	(* Flags to trigger the alarms/events *) //--------------------------------------------------------------------
	
	aSolventLowLevel	 : ARRAY[1..4] OF BOOL; //Flags to check the solvent levels before going to auto cycle
	aSolventNearLowLevel : ARRAY[1..4] OF BOOL; //Flags to warning if the solvent levels are near low level
	bWasteHighLevel		 : BOOL; //Flag to check waste reservoir level before going to auto cycle
	bWasteNearHighLevel	 : BOOL; //Flag to warning if waste reservoir is new high level
	
	bPumpsEStopTriggered : BOOL; //Flag when pumps were running and a emergency stop is triggered
	
	rDiskUsage_C : LREAL;   // % Percentage usage of C: on IPC hard drive
	
	bTCPCLientConnectError	: BOOL; // TCP Client FB_SocketConnect error Flag
	bTCPCLientSendError		: BOOL; // TCP Client FB_SocketSend error Flag
	bTCPCLientReceiveError	: BOOL; // TCP Client FB_SocketReceive error Flag
	bTCPCLientCloseError	: BOOL; // TCP Client FB_SocketCloseAll or FB_SocketClose error Flag
 
	bInvalidSolventSelection : BOOL; // Calibration Invalid Solvent Selection Error
	sStartCalibrationBlockedReason : STRING(255); // Calibration Invalid Solvent Selection Reason
	
	(* Motion Timeouts *) //---------------------------------------------------------------------------------------
	//System Init
	bMotionResetTimeout		: BOOL;	// Motion Timeout during Reset step on PRG_SystemInit
	bMotionEnableTimeout	: BOOL; // Motion Timeout during Enable step on PRG_SystemInit
	bMotionHomeTimeout		: BOOL; // Motion Timeout during Homing step on PRG_SystemInit
	bMotionMoveAbsTimeout	: BOOL; // Motion Timeout during Move Absolute step on PRG_SystemInit
	
	sMotionResetTimeoutAxis		: STRING(64); // String including the axis names to be part of alarm text - Motion Timeout during Reset step on PRG_SystemInit
	sMotionEnableTimeoutAxis	: STRING(64); // String including the axis names to be part of alarm text - Motion Timeout during Enable step on PRG_SystemInit
	sMotionHomeTimeoutAxis		: STRING(64); // String including the axis names to be part of alarm text - Motion Timeout during Homing step on PRG_SystemInit
	sMotionMoveAbsTimeoutAxis	: STRING(64); // String including the axis names to be part of alarm text - Motion Timeout during Move Absolute step on PRG_SystemInit
	
	(* Secondary Functions *) //---------------------------------------------------------------------------------------
	bCalJsonCreationError		: BOOL;		// Error during calibration json file creation
	nCalJsonCreationErrorId		: UDINT;	// Error number ID during calibration json file creation
	
END_VAR

// ---- GVLs/GVL_Calibration.TcGVL
{attribute 'qualified_only'}
VAR_GLOBAL
	
	aCalibPumps         : ARRAY[1..10] OF ST_CalibrationPump;
    bStartCalibration   : BOOL;
    bAbortCalibration   : BOOL;
    bCalibrationRunning : BOOL;
    bCalibrationDone    : BOOL;
    eCalibSolvent       : E_SolventType;
    tDelayStart         : TIME;
    bPrintWhenComplete  : BOOL;
    sGlobalStatus       : STRING[100];
	iPercentLoadBar     : UINT;
	iReplicatesSetpoint : UINT := 1; 
	rAcceptanceCriteria	: LREAL;
	iAllowableFailures	: UINT := 2;
	fbScaleDevice		: FB_ScaleDevice; //Scale Instance Object
	iResultIndex	 	: INT;		 	// Array index on calibration results
	
	aCalibLinearPumps	: ARRAY[1..10] OF ST_LinearPumpCalibration;
	eLeakTestState 		: E_LeakTestState	:= E_LeakTestState.IDLE;
	
	// temp 
	aDosingResults		: ARRAY[1..50] OF ST_DosingResults;
	
	//aCalibCheckResult	: ARRAY[1..100] OF ST_CalibrationPumpResult;
	
	(* Calibration Report*)// -----------------------------------------------------------------------------------------------
	//																													 	|
	stPumpCalReportInfo 	: ST_ReportInfo;	  	//																	  	|
	stPumpCalibrationInfo 	: ST_CalibrationInfo;	//																		|
	stPumpCalibrationData 	: ARRAY[1..250] OF ST_CalibrationData;	//
	//																	
	stLinearCalibrationData : ARRAY[1..10] OF ST_LinearPumpControllDB; // Linear Calibration changing position data from HMI
	//																														|		
	bStartCreationCalJson	: BOOL; // Flag to start the Json creation														|
	bCreationCalJsonDone	: BOOL; // Flag to indicate Json was created Correctly											|
	bCreationCalJsonError	: BOOL; // Flag to indicate Error on Json creation												|
	//																														|
	(**)//-------------------------------------------------------------------------------------------------------------------
	
	//Dosing Procedure
	bDosingTestEnable : BOOL := FALSE;
	
END_VAR

// ---- GVLs/GVL_Constant.TcGVL
{attribute 'qualified_only'}
VAR_GLOBAL CONSTANT

(*Calibration Reports Info*) //----------------------------------------------------------------------------------------------------------------------------
sPumpCalibrationReportName		: STRING(64) := 'Tegan Automated Sample Recovery System (ASRS)';
sPumpCalibrationReportSubName	: STRING(64) := 'Pump Calibration Report';
sSystemID						: STRING(16) := '0001';
sDatabaseName					: STRING(16) := 'ASRS_25';

(*Solvents Types into screen combo boxes*) //--------------------------------------------------------------------------------------------------------------
aSolventsAvailable : ARRAY[1..5] OF STRING := [ 'Solvent 1' , 'Solvent 2', 'Solvent 3', 'Solvent 4', 'Solvent 5' ];

(*IO Screen Texts and pages*) //---------------------------------------------------------------------------------------------------------------------------
aIOPageStarts : ARRAY[0..20] OF UDINT  := [ 0, 1, 3, 5, 7, 9, 11, 13, 15, 17, 19, 21, 23, 25, 27, 29, 31, 33, 35, 37, 40];

aIOList		  :	ARRAY[0..42] OF STRING := [	'  System Overview',
											'  Beckhoff C6030-0060 | Ultra-Compact Industrial PC',
											'  Beckhoff CP2921-0000 | Multi-touch Built-in Control Panel',
											'  Term 1 : EK1100 | EtherCAT Coupler',
											'  Term 2 : EL6070-0033 | License Key Terminal for TwinCAT 3.1',
											
											'  Term 3 : EL6910 | TwinSAFE PLC Module',
											
											'  Term 4 : EL1918 | 8-Channel Digital Input Terminal, TwinSAFE',
											'  Term 5 : EL1918 | 8-Channel Digital Input Terminal, TwinSAFE',
											'  Term 6 : EL1918 | 8-Channel Digital Input Terminal, TwinSAFE',
											
											'  Term 7 : EL2904 | 4-Channel Digital Output Terminal, TwinSAFEE',
											'  Term 8 : EL2904 | 4-Channel Digital Output Terminal, TwinSAFE',
											
											'  Term 9 : EL1809 | 16-Channel Digital Input Terminal',
											'  Term 10: EL2809 | 16-Channel Digital Output Terminal',
											
											'  Term 11: EL2624 | 4-channel Relay Output Terminal',
											
											'  Term 12: EL9410 | Power supply terminal for E-bus, with diagnostics',
											'  Term 13: EL3058 | 8-channel analog input, current, single-ended',
											'  Term 14: EL9576 | Brake chopper terminal',
											'  Term 15: EL7211-9014 | 1-channel Motion interface, servomotor',
											'  Term 16: EL7211-9014 | 1-channel Motion interface, servomotor',
											'  Term 17: EL3022 | 2-channel analog input, current, differential',
											'  Term 18: EL1809 | 16-channel digital input, 24 V DC, 3 ms',
											'  Term 19: EL2904 | 4-Channel Digital Output Terminal, TwinSAFE',
											'  Term 20: EL6631 |  2-port Communication PROFINET RT Interface',					
											
											'  Term 22: EL7062 | 2-channel Motion Stepper Motor Interface',
											'  Term 23: EL7062 | 2-channel Motion Stepper Motor Interface',
											'  Term 24: EL7062 | 2-channel Motion Stepper Motor Interface',
											'  Term 25: EL7062 | 2-channel Motion Stepper Motor Interface',
											'  Term 26: EL7062 | 2-channel Motion Stepper Motor Interface',
											'  Term 27: EL7062 | 2-channel Motion Stepper Motor Interface',
											'  Term 28: EL7062 | 2-channel Motion Stepper Motor Interface',
											'  Term 29: EL7062 | 2-channel Motion Stepper Motor Interface',
											'  Term 30: EL7062 | 2-channel Motion Stepper Motor Interface',
											'  Term 31: EL7062 | 2-channel Motion Stepper Motor Interface',
											'  Term 32: EL7062 | 2-channel Motion Stepper Motor Interface',
											'  Term 33: AX8101 | Single-axis Module',
											
											'  BOX 01  - AL1333 | IO-Link master with EtherCAT interface',
											'  BOX 02 - AMI8100 | Compact Integrated Servo Drives',	
											'  BOX 03 - AMI8100 | Compact Integrated Servo Drives',		
											'  BOX 04 - AMI8100 | Compact Integrated Servo Drives',
											'  BOX 05 - AMI8100 | Compact Integrated Servo Drives',	
											'  BOX 06 - AMI8100 | Compact Integrated Servo Drives'			
											];

//Naming the axis by index for alarms text assemble
sMotionText	: ARRAY[1..28] OF STRING(5) := [ 'M1,',
											 'M2,',
											 'M3,',
											 'V1,',
											 'V2,',
											 'V3,',
											 'V4,',
											 'V5,',
											 'LP1,',
											 'LP2,',
											 'LP3,',
											 'LP4,',
											 'LP5,',
											 'LP6,',
											 'LP7,',
											 'LP8,',
											 'LP9,',
											 'LP10,',
											 'RP1,',
											 'RP2,',
											 'RP3,',
											 'RP4,',
											 'RP5,',
											 'RP6,',
											 'RP7,',
											 'RP8,',
											 'RP9,',
											 'RP10,'
 											];


(* ----------------------------------------------------------------------------------- HMI COLORS ----------------------------------------------------------------------------------- *)
	
    sWHITE                              :   STRING(40)  := '{"color":"rgba(255,255,255,255)"}';
    sBLACK                              :   STRING(40)  := '{"color":"rgba(0,0,0,1)"}';
    sYELLOW                             :   STRING(40)  := '{"color":"rgba(255,255,0,1)"}';
    sGREEN                             	:   STRING(40)  := '{"color":"rgba(70,166,63,1)"}';
	sLGREEN                             :   STRING(40)  := '{"color":"rgba(58,211,20,1)"}';
    sORANGE                             :   STRING(40)  := '{"color":"rgba(255,153,51,1)"}';
    sNYPROORANGE                        :   STRING(40)  := '{"color":"rgba(255,140,0,1)"}';
    sRED                                :   STRING(40)  := '{"color":"rgba(255,0,0,1)"}';
	sLRED                               :   STRING(40)  := '{"color":"rgba(233,53,44,1)"}';
    sBLUE                               :   STRING(40)  := '{"color":"rgba(0,0,255,1)"}';
	sLBLUE                              :   STRING(40)  := '{"color":"rgba(0,162,232,1)"}';
    sGREY                               :   STRING(40)  := '{"color":"rgba(164,158,158,1)"}';
    sScreenGREY                         :   STRING(40)  := '{"color":"rgba(225,225,225,1)"}';
    sDARKGREY                           :   STRING(40)  := '{"color":"rgba(50,50,50,1)"}';
    sPURPLE                             :   STRING(40)  := '{"color":"rgba(128,0,128,1)"}';
    sVIOLET                             :   STRING(40)  := '{"color":"rgba(204,153,255,1)"}';
    sTRANSP                             :   STRING(40)  := '{"color":"rgba(255,255,255,0)"}';
    sGREENPass                          :   STRING(40)  := '{"color":"rgba(0,153,51,1)"}';
    sREDFail                            :   STRING(40)  := '{"color":"rgba(244,68,68,255)"}';
    sBLUEInProgress                     :   STRING(40)  := '{"color":"rgba(54,100,221,1)"}';
	sGREENISHTEAColor					:	STRING(40)  := '{"color":"rgba(60,192,134,255)"}'	;		

	nBLACK								: 	DWORD 	:= 	16#FF000000;	 // format: TTRRGGBB where T -> 00 = full transparency and FF = full opaque
	nWHITE								: 	DWORD 	:= 	16#FFFFFFFF;
	nYELLOW								: 	DWORD 	:= 	16#FFFFFF00; 
	nGREEN								: 	DWORD 	:= 	16#FF008A00;
	nLIGHTGREEN                         :   DWORD   :=  16#FF98FB89;
	nORANGE								: 	DWORD 	:= 	16#FFFFA500;
	nNYPROORANGE						:	DWORD	:=	16#FFF05322;
	nRED								: 	DWORD 	:= 	16#FFFF0000;
	nBLUE								: 	DWORD 	:= 	16#FF0000FF;
	nLIGHTBLUE                          :   DWORD   :=  16#FF08ADF4;
	nGREY								: 	DWORD 	:= 	16#FFA9A9A9;	
	nDARKGREY							:	DWORD	:=	16#FF808080;
	nPURPLE								:	DWORD	:=	16#FF800080;
	nVIOLET								:	DWORD	:=	16#FFEE82EE;
	nTRANSP								:	DWORD	:=	16#00FFFFFF;	// full transparent WHITE
	
(* ----------------------------------------------------------------------------------- HMI COLORS ----------------------------------------------------------------------------------- *)
											
END_VAR

// ---- GVLs/GVL_HMI.TcGVL
{attribute 'qualified_only'}
{attribute 'TcHmiSymbol' := 'true'}
VAR_GLOBAL
	
	//Info Screen
	stInfo				: ST_InfoPage; 	// Project Info screen details to be shown on HMI
	stReminders 		: ST_Reminders; // Reminders screen signals to be shown on HMI
	
	HMIDigInputs		 : ST_HMIDigInputs;  //Digital Inputs data from HMI
	HMIDigOutputs		 : ST_HMIDigOutputs; //Digital Outputs data for HMI

	HMIAnimation		 : ST_HMIAnimation; //Variables needed to animate the HMI
	bHMICalibrationBox	 : BOOL; 			//Calibration Box presence
	
	eMachineMode		 : E_MachineMode; //Machine mode selection from HMI
	
	bIncoherenceDetected : BOOL := FALSE; //Incoherence Monitoring that could block master controll to enter in autoCycle
	bIncoherenceAlert	 : BOOL := FALSE; //Incoherence alert to show an alert on HMI. Event trigger DesktopView 
	
	sDateAndTimeEventTriggered	: STRING(256); //Linear Pumps save procedure gets the date and time from hmi
	sUserNameEventTriggered		: STRING(256); //Linear Pumps save procedure gets the hmi username
	
	sActivatedRecipeHomeNaming  : STRING(256); // Recipe name shown on home screen when a recipe is active
	
	(* Auto Cycle Popup *) // ---------------------------------------------------------------------------------------------------------------------------------
	sAutoCycleComment			: STRING(256); // Comment inserted by user before going to autocycle
	bStartAutoCycleButton		: BOOL := FALSE; // Start AUto Cycle Button from Auto Cycle popup
	bShowAutoCyclePopup     	: BOOL := FALSE; // Controls Auto Cycle popup visibility on HMI
	bSystemReady_ReqAutoCycle 	: BOOL := FALSE; // One-shot request to go to AUTO_CYCLE from SystemReady
	
	// --- Auto cycle soft-stop / hold control ---
    bAutoCycleHoldReq        : BOOL	:= FALSE;  // 1st STOP inside AUTO_CYCLE
    bAutoCycleHoldActive     : BOOL	:= FALSE;  // TRUE while StateMachine is in PAUSE_STATE
    bAutoCycleHoldPopup      : BOOL := FALSE;  // HMI shows the "Cancel / Continue" popup
	bAutoCyclePrimeSolvents	 : BOOL	:= FALSE;  // HMI flag for prime the solvents used on auto cycle before metering the rinse

    bAutoCycleContinueCmd    : BOOL	:= FALSE;  // HMI "Continue" button
    bAutoCycleCancelCmd      : BOOL	:= FALSE;  // HMI "Cancel Run" button
	
	bLightsToggleButton	 : BOOL := FALSE; // Home screen toggle button for turn lights on or off on HMI 
	rTimeCountingDown 	 : LREAL; 		  //Countdown time for shutdown or rebooting PLC
	sCountdownPopupText	 : STRING(16);	  //Countdown Popup text for shutdown or rebooting PLC
	
	//Machine Mode Blinking
	bMachineModeBlinking : BOOL := FALSE;	// Flashing variable to blink the state on HMI headbar
	bMachineModeScan	 : BOOL := FALSE;	// Flashing variable to scan some controls on HMI home screen
	bHomeScreenLoaded	 : BOOL := FALSE;	// Flag to tell when the home screen is loaded or not
	
	//User Management
	stUserMgmtHistoryEvent  : ST_UserMgmtHistoryEvent;
	stUsers          		: ARRAY[1..50] OF ST_User;  // users list | max 50 users
    iLoggedUserID    		: INT := -1;                // -1 = no one logged in
    dtCurrentLogin   		: DT;
    tSessionStart    		: TIME;

	// <Recipe> Variables needed to handle recipe --------------------------------------------------------------------------------------------------------------
	aAvailableFiles         : ARRAY[0..99] OF ST_RecipeFileInfo;
    iFileCount              : INT;
	
    bRefreshRecipeList      : BOOL; 			//List the recipe files from HMI
    bRecipeLoadFromFile	 	: BOOL := FALSE; 	//load recipe button from HMI
	bReloadRecipeDatagrids	: BOOL := FALSE;	//Reload the recipe in stCurrentRecipe to the datagrids if the cancel button is pressed when creating new recipe
    sSelectedRecipeName     : STRING(255); 		// Selected name from hmi list popup
	bRecipeCorrectLoaded	: BOOL; 			// Flag to identify if there is a recipe loaded to proceed with the recovery
	bRecipeLoadFailed		: BOOL; 			// Flag to identify if there was any error loading the recipe file
	
	bRecipeActivateButton	: BOOL := FALSE; // Activate Recipe command from recipe activate button 
	bRecipeActivateDone		: BOOL := FALSE; // Activate done flag after command from recipe activate button
	bRecipeActivateError	: BOOL := FALSE; // Activate Error flag after command from recipe activate button
	
	bRecipeSaveButton		: BOOL := FALSE; // save command from recipe save button
	bRecipeSaveDone			: BOOL := FALSE; // Save done flag after save command from recipe save button
	bRecipeSaveError		: BOOL := FALSE; // Save Error flag after save command from recipe save button
	
	stDeleteRecipeInfo		: ST_RecipeFileInfo;
	bDeleteRecipeButton		: BOOL := FALSE; // Delete recipe button Action - Open delete popup
	bDeleteRecipeConfirm	: BOOL := FALSE; // Delete recipe confirmation action
	bDeleteRecipeError		: BOOL := FALSE; // Delete recipe Error flag
	bDeleteRecipeDone		: BOOL := FALSE; // Delete recipe done flag
	
	bNewRecipeButton		: BOOL := FALSE; // New Recipe button on recipe screen.
	
	//Recipe HMI View - data needs to be transposed for better view and handled by HMI
	stRecipeInfo		 : ST_RecipeInfo;	// Recipe info datagrid showed on HMI
	aSolventAndTimesRows : ARRAY[1..3] OF ST_HMI_SolventAndTimeRow;	// Recipe Solvent And Times transposed datagrid showed on HMI
	aVolumeRows 		 : ARRAY[1..10] OF ST_HMI_VolumesRow; 		// Recipe Volumes transposed datagrid showed on HMI
	aOtherParamsRows 	 : ARRAY[1..8] OF ST_HMI_OtherParamsRow;	// Recipe Other Parameters transposed datagrid showed on HMI
	// <\Recipe> -----------------------------------------------------------------------------------------------------------------------------------------------
	
	// <Calibration> Variables needed to handle calibration tasks from HMI -------------------------------------------------------------------------------------
	
	bCalLeakTestButton		: BOOL := FALSE; // Leak test action button from HMI
	bCalLeakTestPass		: BOOL := FALSE; // Leak test passed flag
	bCalLeakTestFail		: BOOL := FALSE; // Leak test failed flag
	bCalLeakTestError		: BOOL := FALSE; // Leak test error flag
	rCalLeakTestPressure	: LREAL;		 // Leak test pressure reading from sensor
	
	bCalPressureUpSystemBt	: BOOL := FALSE; // HMI Button responsible for pressurize the system
	bCalHoldSysPressureBt	: BOOL := FALSE; // HMI Button responsible for shut the air off the system
	bCalStopLeakTestBt		: BOOL := FALSE; // HMI Button responsible for stopping the leak test
	
	bCalLinearPumpsEnableBt	: BOOL := FALSE; // Linear pumps Enable motors button
	bCalLinearPumpsHomeBt	: BOOL := FALSE; // Linear pumps Homing motors button
	bCalLinearPumpsMoveBt	: BOOL := FALSE; // Linear pumps Move motors button
	bCalLinearPumpsStopBt	: BOOL := FALSE; // Linear pumps Stop motors button
	bCalLinearPumpsSaveBt	: BOOL := FALSE; // Linear pumps Save Parameters button
	bCalLinearPumpsDirty	: BOOL := FALSE; // flag to indicate when there was any change on the linear pumps.
	
	bStartCalibrationBt		: BOOL := FALSE; //Start Calibration Bt from HMI
	bAbortCalibrationBT		: BOOL := FALSE; //Abort Calibration Bt from HMI
	
	aCalibPumps         	: ARRAY[1..10] OF ST_CalibrationPump;		// Calibration rotary Pumps settings
	aCalibLinearPumps		: ARRAY[1..10] OF ST_LinearPumpCalibration; // Calibration linear Pumps settings
	aCalPumpResults    		: ARRAY[1..10] OF ST_CalibrationPumpResult; // Rotary Pumps result structure
	
	iSelectedCalibrationSolvent : USINT := 0; // Solvent Selection - 0 = None, 1 = Solvent 1, 2 = Solvent 2, etc.
	
	rLinearPumpsLastAdjustUser	: STRING(128);		 // Linear pumps last adjusted username
	rLinearPumpsLastAdjustDate	: DATE;				 // Linear pumps last adjusted Date
	
	bScaleNeedsAtention		: BOOL := FALSE; // Flag to trigger a popup on hmi telling operator to handle the scale error | Listener on Desktop.view Index Region
	bScaleFixed				: BOOL := FALSE; // Feedback from hmi to tell the system that scale is ready to continue
	
	bCalBoxNeedsAttention	: BOOL := FALSE; // Flag to trigger a popup on hmi telling operator to fill up the calibration box
	bCalBoxFixed			: BOOL := FALSE; // Feedback from hmi to tell the system that the calibration box is ready to continue
	
	bCalMoveValves			: BOOL  := FALSE; // Manual Valves Movement from calibration screen 
	iCalMoveValvesPosition	: USINT := 1; 	  // Manual Valves Position from calibration screen 
	bCalMoveM1Motor			: BOOL  := FALSE; // Manual M1 Motor Movement from calibration screen 
	iCalMoveM1MotorPosition	: USINT := 1; 	  // Manual M1 Motor Position from calibration screen 
	
	sCalLeakTestStatus		: STRING(32);	  // Automatic sealing test status text on calibration screen 
	iCalLeakTestState		: USINT := 1;	  // Automatic sealing test image state LED on calibration screen 
	
	//UILoadBar
	bCalibStepLoading   : BOOL;		  	// Loadbar progress enable variable on calibration screen
    rCalibStepPercent   : REAL;       	// Loadbar progress for step time on calibration screen [0..100]
    sCalibProgressLabel : STRING(80);	// Loadbar progress label on calibration screen
	
	// <\Calibration> ------------------------------------------------------------------------------------------------------------------------------------------
	
	// <Reports Listing> ---------------------------------------------------------------------------------------------------------------------------------------
	
	aCalibrationReportList      : ARRAY[1..100] OF ST_CalibrationReportListItem;
    stSelectedCalibReportHeader : ST_CalibrationReportHeader;
    aSelectedCalibReportLines   : ARRAY[1..300] OF ST_CalibrationReportLine;

    sSelectedReportId           : STRING(50);

    bLoadCalibrationReportList  : BOOL;
    bLoadSelectedCalibReport    : BOOL;
    bSelectedReportReady        : BOOL;
    bReportListReady            : BOOL;
    bReportQueryBusy            : BOOL;
    bReportQueryError           : BOOL;
	
	aReportSearchResult : ARRAY[1..100] OF ST_ReportListItem;
	uiReportSearchCount : UDINT;
	eSelectedReportType : E_ReportType;
	sSelectedPrimaryID  : STRING(50);
	dtDateFrom          : STRING(30);
	dtDateTo            : STRING(30);
	
	// <Machine Settings> Variables to handle solvents insert in the settings screen ----------------------------------------------------------------------------
	HMIParameters		 : ST_HMIParameters; 					// Motion Parameters from HMI inputs
	stHMICalibParameters : ST_CalibrationSettings;				// Calibration Parameters from HMI inputs
	stHMIPumpParameters	 : ST_PumpSettings;						// Pump Parameters from HMI inputs
	stLeakTestParameters : ST_LeakTestSettings;					// Leak Test Parameters from HMI Inputs
	stHMISolventsInfo	 : ARRAY[1..4] OF ST_SolventsSettings;	// Solvents name and density to be inserted on the settings screen 		
	bReloadHMIParameters : BOOL := FALSE;						// Reload parameters from GVL_Settings when first loading the screen
	bSaveParametersBt	 : BOOL := FALSE; 						// Save Parameters from HMI
	bSaveParametersDone	 : BOOL := FALSE;						// Save Parameters Done flag from PLC
 	bSaveParametersError : BOOL := FALSE;						// Save Parameters Error flag from PLC
	bSaveSolventsBt		 : BOOL := FALSE;						// Save Solvents change from HMI settings screen
	bSaveSolventsDone	 : BOOL := FALSE;						// Save Solvents Done flag from HMI settings screen
	bSaveSolventsError	 : BOOL := FALSE;						// Save Solvents Error flag from HMI settings screen
	
	(* Manual Motors Moviment *) //--------------------------------------------------------------------------------------------------------------
	ManualMov			: ST_MotorsJog; // Manual Joging motors from old manual screen
	
	aManualMotorsCmd 	: ARRAY[1..3] OF ST_MotorCommand;	// Manual Motors commands from manual screen
    aManualValvesCmd 	: ARRAY[1..5] OF ST_ValveCommand;	// Manual Valves commands from manual screen
    aManualPumpsCmd  	: ARRAY[1..10] OF ST_PumpCommand;	// Manual Pumps commands from manual screen
	
	bRunPumpsBySpeedBt 		: BOOL;	// Button Run pumps by Speed from manual screen
	bRunPumpsByVolumeBt 	: BOOL;	// Button Run pumps by Volume from manual screen
	bRunPumpsByDistanceBt 	: BOOL;	// Button Run pumps by Distance from manual screen
	bStopPumpsBt 			: BOOL;	// Button Stop pumps movememnt from manual screen
	
	(* Alarms and Events triggers from HMI JS Trigger*) //-------------------------------------------------------------------------------------------------------------
	bM1MoveNotAllowedTrigger	: BOOL;	// 'IE-100: M1 Movement Not allowed'; (* JS from Run M1 Button - Manual screen *)
	bM2MoveNotAllowedTrigger	: BOOL;	// 'IE-100: M2 Movement Not allowed'; (* JS from Run M2 Button - Manual screen *)
	bM3MoveNotAllowedTrigger	: BOOL;	// 'IE-101: M3 Movement Not allowed'; (* JS from Run M3 Button - Manual screen *)
	bCalNotAllowedTrigger		: BOOL;	// 'IE-110: Attempt to perform a calibration procedure without a calibration box'; (* JS from Start Calibration Button - Calibration screen *)
		
	// <IO Screen> Variables for IO Screen use (*-----------------------------------------------------------------------------------------------)
	
	nSelectedIO		: UDINT; // Selection made by IO screen combobox
	
	aIOTerm04		: ARRAY[1..8] OF BOOL;
	aIOTerm05		: ARRAY[1..8] OF BOOL; 
	aIOTerm06		: ARRAY[1..8] OF BOOL; 
	aIOTerm07		: ARRAY[1..4] OF BOOL; 
	aIOTerm08		: ARRAY[1..4] OF BOOL;
	aIOTerm09		: ARRAY[1..16] OF BOOL;
	aIOTerm10		: ARRAY[1..16] OF BOOL;
	aIOTerm11		: ARRAY[1..4] OF BOOL;   
	aIOTerm12		: ARRAY[1..2] OF BOOL;
	aIOTerm13		: ARRAY[1..8] OF REAL;
	aIOTerm14		: ARRAY[1..8] OF BOOL;
   	iIOTerm14DCIn	: UDINT;
	aIOTerm15		: ARRAY[1..3] OF BOOL;
	aIOTerm15Values : ARRAY[1..3] OF LREAL;
	iIOTerm15ErrorCode	: UDINT;
	aIOTerm16		: ARRAY[1..3] OF BOOL;
	aIOTerm16Values : ARRAY[1..3] OF LREAL;
	iIOTerm16ErrorCode	: UDINT;
	aIOTerm17		: ARRAY[1..6] OF BOOL;
	aIOTerm17Values : ARRAY[1..2] OF LREAL;
	aIOTerm18		: ARRAY[1..16] OF BOOL;
	aIOTerm19		: ARRAY[1..4] OF BOOL; 
	stIOTerm23		: ST_EL7062IOInfo;
	stIOTerm24		: ST_EL7062IOInfo;
	stIOTerm25		: ST_EL7062IOInfo;
	stIOTerm26		: ST_EL7062IOInfo;
	stIOTerm27		: ST_EL7062IOInfo;
	stIOTerm28		: ST_EL7062IOInfo;
	stIOTerm29		: ST_EL7062IOInfo;
	stIOTerm30		: ST_EL7062IOInfo;
	stIOTerm31		: ST_EL7062IOInfo;
	stIOTerm32		: ST_EL7062IOInfo;
	stIOTerm34		: ST_AX8101IOInfo;
	aIOBox1			: ARRAY[1..8] OF REAL;
	aIOAMI8000		: ARRAY[1..5] OF ST_AMI8000IOInfo;
	
	// <\IO Screen>  (*-------------------------------------------------------------------------------------------------------------------------)
	
	//TEMP
	bResetM1MotorBt : BOOL := FALSE; // Temporary Motor M1 Reset button on old joging manual screen while new motor is not installed
	
	// UserManagement -------------------------------------------------------------------------------------------------------------------
	
	passwordOk: BOOL;
	
END_VAR

// ---- GVLs/GVL_IO.TcGVL
{attribute 'qualified_only'}
VAR_GLOBAL
	
	(* IO used in the software *) //----------------------------------------------------------------------------------------
	gDigInputs	 		AT%I*	:	ST_EL1809;	//Digital inputs at Terminals 21 and 30 [EL1809]
	gDigOutputs			AT%Q*	:	ST_EL2809;	//Digital Outputs at Terminal 22 		[EL2809]
	gRelayOutputs		AT%Q*	:	ST_EL2624;	//Digital Relay Outputs at Terminal 23 	[EL2624]
	gAnalogInputs		AT%I*	:	ST_EL3058; 	//Analog inputs at Terminals 25 		[EL3058]
	gAnalogInputs2Ch	AT%I*	:	ST_EL3022;	//Analog inputs at Terminals 17 		[EL3022]
	gProfinetInput		AT%I*	:	ST_EL6631;  //Profinet inputs by Device 5 			[EL6631]
	
	gParameters			: ST_HMIParameters; 	//Machine Parameters
	gSetSolenoidControl : FB_SetSolenoid;		//FB only instance to control solenoids valves set. 
	
	// Safety Alias
	bInAckSignal		AT %I* : BOOL; // Aknowledge input
	bInResetSignal		AT %Q* : BOOL; // Reset input
	
	stEL6910	: ST_EL6910; // Safety PLC - Terminal 3
	
	// Is Vials Rack Present?
	bVialRackPresent : BOOL;
	
	// power source signal for recovery valves position purposes
	bPowerSupplyDropSignal	: BOOL := FALSE;
	
	//----------------------------------------------------------------------------------------------------------------------
	// IO Terminals to feed HMI IO Screens
	//----------------------------------------------------------------------------------------------------------------------
	
	// TERMINAL - EK1100 EtherCAT Coupler (Term 1)
	nEK1100T01State		AT %I*	: UINT;	//Terminal State from IO Terminal Info Data	
	bEK1100T01State				: BOOL; //Control flag from terminal state	
	sEK1100T01Status			: STRING(200);
	
	// TERMINAL - EK1100 EtherCAT Coupler (Term 22)
	nEK1100T22State		AT %I*	: UINT;	//Terminal State from IO Terminal Info Data
	bEK1100T22State				: BOOL; //Control flag from terminal state	
	sEK1100T22Status			: STRING(200);	
	
	// TERMINAL - EL6070-0033	License Key Terminal for TwinCAT 3.1 (Term 2)
	nEL6070State		AT %I*	: UINT;	// EL6070-0033 State from IO Terminal Info Data	
	bEL6070State				: BOOL; //Control flag from terminal state	
	sEL6070Status				: STRING(200);	
	
	// TERMINAL - EL1918 Safety Inputs (Term 4)
	nEL1918T04State		AT %I*	: UINT;	// EL1918 State from IO Terminal Info Data
	bEL1918T04State				: BOOL; //Control flag from terminal state		
	sEL1918T04Status			: STRING(200);	
	
	// TERMINAL - EL1918 Safety Inputs (Term 5)
	nEL1918T05State		AT %I*	: UINT;	// EL1918 State from IO Terminal Info Data
	bEL1918T05State				: BOOL; //Control flag from terminal state		
	sEL1918T05Status			: STRING(200);

	// TERMINAL - EL1918 Safety Inputs (Term 6)
	nEL1918T06State		AT %I*	: UINT;	// EL1918 State from IO Terminal Info Data	
	bEL1918T06State				: BOOL; //Control flag from terminal state	
	sEL1918T06Status			: STRING(200);	
	
	// TERMINAL - EL2904 Safety Outputs (Term 7)
	nEL2904T07State		AT %I*	: UINT;	// EL2904 State from IO Terminal Info Data
	bEL2904T07State				: BOOL; //Control flag from terminal state		
	sEL2904T07Status			: STRING(200);
	
	// TERMINAL - EL2904 Safety Outputs (Term 8)
	nEL2904T08State		AT %I*	: UINT;	// EL2904 State from IO Terminal Info Data	
	bEL2904T08State				: BOOL; //Control flag from terminal state	
	sEL2904T08Status			: STRING(200);
	
	// TERMINAL - EL1809 Digital Inputs (Term 9)
	nEL1809T09State		AT %I*	: UINT;	// State from IO Terminal Info Data	
	bEL1809T09State				: BOOL; // Control flag from terminal state	
	sEL1809T09Status			: STRING(200);
	
	// TERMINAL - EL2809 Digital Outputs (Term 10)
	nEL2809T10State		AT %I*	: UINT;	// State from IO Terminal Info Data	
	bEL2809T10State				: BOOL; // Control flag from terminal state	
	sEL2809T10Status			: STRING(200);
	
	// TERMINAL - EL2624 Relay Outputs (Term 11)
	nEL2624T11State		AT %I*	: UINT;	// State from IO Terminal Info Data	
	bEL2624T11State				: BOOL; // Control flag from terminal state	
	sEL2624T11Status			: STRING(200);
	
	// TERMINAL - EL9410 Power Supply (Term 12)
	nEL9410T12State		AT %I*	: UINT;	// State from IO Terminal Info Data	
	bEL9410T12State				: BOOL; // Control flag from terminal state	
	sEL9410T12Status			: STRING(200);
	bEL9410UPStatus		AT %I*	: BOOL; // Terminal UP Status
	bEL9410USStatus		AT %I*	: BOOL; // Terminal US Status
	
	// TERMINAL - EL3058 Relay Outputs (Term 13)
	nEL3058T13State		AT %I*	: UINT;	// State from IO Terminal Info Data	
	bEL3058T13State				: BOOL; // Control flag from terminal state	
	sEL3058T13Status			: STRING(200);
	
	// TERMINAL - EL9576 Relay Outputs (Term 14)
	nEL9576T14State			AT %I*	: UINT;	// State from IO Terminal Info Data	
	bEL9576T14State					: BOOL; // Control flag from terminal state	
	sEL9576T14Status				: STRING(200);
	bEL9576T14Overtemp		AT %I*	: BOOL;
	bEL9576T14I2TError		AT %I*	: BOOL;
	bEL9576T14I2TWarning	AT %I*	: BOOL;
	bEL9576T14OverVoltage	AT %I*	: BOOL;
	bEL9576T14UnderVoltage	AT %I*	: BOOL;
	bEL9576T14ChopperOn		AT %I*	: BOOL;
	bEL9576T14OverCurrent	AT %I*	: BOOL;
	bEL9576T14DCLinkVoltage	AT %I*	: UDINT;
	
	// TERMINAL - EL7211 Relay Outputs (Term 15)
	nEL7211T15State				: UINT;	// State from IO Terminal Info Data	
	bEL7211T15State				: BOOL; // Control flag from terminal state	
	sEL7211T15Status			: STRING(200);
	
	// TERMINAL - EL7211 Relay Outputs (Term 16)
	nEL7211T16State				: UINT;	// State from IO Terminal Info Data	
	bEL7211T16State				: BOOL; // Control flag from terminal state	
	sEL7211T16Status			: STRING(200);
	
	// TERMINAL - EL3022 Relay Outputs (Term 17)
	nEL3022T17State			AT %I*	: UINT;	// State from IO Terminal Info Data	
	bEL3022T17State					: BOOL; // Control flag from terminal state	
	sEL3022T17Status				: STRING(200);
	bEL3022ChAUnderRange	AT %I*	: BOOL; // Control UnderRange flag from terminal ch A
	bEL3022ChAOverRange		AT %I*	: BOOL; // Control OverRange flag from terminal ch A
	bEL3022ChAError			AT %I*	: BOOL; // Control Error flag from terminal ch A
	bEL3022ChBUnderRange	AT %I*	: BOOL; // Control UnderRange flag from terminal ch B
	bEL3022ChBOverRange		AT %I*	: BOOL; // Control OverRange flag from terminal ch B
	bEL3022ChBError			AT %I*	: BOOL; // Control Error flag from terminal ch B
	
	// TERMINAL - EL1809 Relay Outputs (Term 18)
	nEL1809T18State		AT %I*	: UINT;	// State from IO Terminal Info Data	
	bEL1809T18State				: BOOL; // Control flag from terminal state	
	sEL1809T18Status			: STRING(200);
	
	// TERMINAL - EL2904 Safety Outputs (Term 19)
	nEL2904T19State		AT %I*	: UINT;	// EL2904 State from IO Terminal Info Data	
	bEL2904T19State				: BOOL; //Control flag from terminal state	
	sEL2904T19Status			: STRING(200);
	
	// TERMINAL - EL2904 Safety Outputs (Term 20)
	nEL6631T20State		AT %I*	: UINT;	// EL2904 State from IO Terminal Info Data	
	bEL6631T20State				: BOOL; //Control flag from terminal state	
	sEL6631T20Status			: STRING(200);
	
	// TERMINAL - EL7062 EtherCAT 2-channel stepper motor interface  (Term 23)
	nEL7062T23State				: UINT;	//Terminal State from IO Terminal Info Data
	bEL7062T23State				: BOOL; //Control flag from terminal state	
	sEL7062T23Status			: STRING(200);	
	
	// TERMINAL - EL7062 EtherCAT 2-channel stepper motor interface  (Term 24)
	nEL7062T24State				: UINT;	//Terminal State from IO Terminal Info Data
	bEL7062T24State				: BOOL; //Control flag from terminal state	
	sEL7062T24Status			: STRING(200);	
	
	// TERMINAL - EL7062 EtherCAT 2-channel stepper motor interface  (Term 25)
	nEL7062T25State				: UINT;	//Terminal State from IO Terminal Info Data
	bEL7062T25State				: BOOL; //Control flag from terminal state	
	sEL7062T25Status			: STRING(200);	
	
	// TERMINAL - EL7062 EtherCAT 2-channel stepper motor interface  (Term 26)
	nEL7062T26State				: UINT;	//Terminal State from IO Terminal Info Data
	bEL7062T26State				: BOOL; //Control flag from terminal state	
	sEL7062T26Status			: STRING(200);	
	
	// TERMINAL - EL7062 EtherCAT 2-channel stepper motor interface  (Term 27)
	nEL7062T27State				: UINT;	//Terminal State from IO Terminal Info Data
	bEL7062T27State				: BOOL; //Control flag from terminal state	
	sEL7062T27Status			: STRING(200);	
	
	// TERMINAL - EL7062 EtherCAT 2-channel stepper motor interface  (Term 28)
	nEL7062T28State				: UINT;	//Terminal State from IO Terminal Info Data
	bEL7062T28State				: BOOL; //Control flag from terminal state	
	sEL7062T28Status			: STRING(200);	
	
	// TERMINAL - EL7062 EtherCAT 2-channel stepper motor interface  (Term 29)
	nEL7062T29State				: UINT;	//Terminal State from IO Terminal Info Data
	bEL7062T29State				: BOOL; //Control flag from terminal state	
	sEL7062T29Status			: STRING(200);	
	
	// TERMINAL - EL7062 EtherCAT 2-channel stepper motor interface  (Term 30)
	nEL7062T30State				: UINT;	//Terminal State from IO Terminal Info Data
	bEL7062T30State				: BOOL; //Control flag from terminal state	
	sEL7062T30Status			: STRING(200);	
	
	// TERMINAL - EL7062 EtherCAT 2-channel stepper motor interface  (Term 31)
	nEL7062T31State				: UINT;	//Terminal State from IO Terminal Info Data
	bEL7062T31State				: BOOL; //Control flag from terminal state	
	sEL7062T31Status			: STRING(200);	
	
	// TERMINAL - EL7062 EtherCAT 2-channel stepper motor interface  (Term 32)
	nEL7062T32State				: UINT;	//Terminal State from IO Terminal Info Data
	bEL7062T32State				: BOOL; //Control flag from terminal state	
	sEL7062T32Status			: STRING(200);	
	
	// TERMINAL - AX8620  (Term 33)
	nAX8620T33State		AT %I*	: UINT;	//Terminal State from IO Terminal Info Data
	bAX8620T33State				: BOOL; //Control flag from terminal state	
	sAX8620T33Status			: STRING(200);	
	
	// TERMINAL - AX8108  (Term 34)
	nAX8108T34State				: UINT;	//Terminal State from IO Terminal Info Data
	bAX8108T34State				: BOOL; //Control flag from terminal state	
	sAX8108T34Status			: STRING(200);	
	
	// Box 1 - Ifm AL1333  (Box 1)
	nAL1333Box1State	AT %I*	: UINT;	//Terminal State from IO Terminal Info Data
	bAL1333Box1State			: BOOL; //Control flag from terminal state	
	sAL1333Box1Status			: STRING(200);
	stAL1333info				: ST_AL1333;	
	
	// Box 8 - AMI8000-0100  (Box 8)
	nAMI8000Box8State			: UINT;	//Terminal State from IO Terminal Info Data
	bAMI8000Box8State			: BOOL; //Control flag from terminal state	
	sAMI8000Box8Status			: STRING(200);
	
	// Box 9 - AMI8000-0100  (Box 9)
	nAMI8000Box9State			: UINT;	//Terminal State from IO Terminal Info Data
	bAMI8000Box9State			: BOOL; //Control flag from terminal state	
	sAMI8000Box9Status			: STRING(200);
	
	// Box 10 - AMI8000-0100  (Box 10)
	nAMI8000Box10State			: UINT;	//Terminal State from IO Terminal Info Data
	bAMI8000Box10State			: BOOL; //Control flag from terminal state	
	sAMI8000Box10Status			: STRING(200);
	
	// Box 11 - AMI8000-0100  (Box 11)
	nAMI8000Box11State			: UINT;	//Terminal State from IO Terminal Info Data
	bAMI8000Box11State			: BOOL; //Control flag from terminal state	
	sAMI8000Box11Status			: STRING(200);
	
	// Box 12 - AMI8000-0100  (Box 12)
	nAMI8000Box12State			: UINT;	//Terminal State from IO Terminal Info Data
	bAMI8000Box12State			: BOOL; //Control flag from terminal state	
	sAMI8000Box12Status			: STRING(200);
	
	//----------------------------------------------------------------------------------------------------------------------
	
END_VAR

// ---- GVLs/GVL_Reports.TcGVL
{attribute 'qualified_only'}
VAR_GLOBAL

(***** Search Screen - Filters / Commands ************************************************)

bSearchRequest          	: BOOL;
bSearchBusy             	: BOOL;
bSearchDone             	: BOOL;
bSearchError            	: BOOL;
bClearSearchScreen 			: BOOL;
bBuildCurrentLinearReport 	: BOOL;
bBuildLastPostRunReport 	: BOOL;
bBuildLastPumpCalibrationReport : BOOL;
sSearchStatus           	: STRING(100);

sDateFromFilter 		: STRING(30);
sDateToFilter   		: STRING(30);
bUseDateFilter  		: BOOL;
bClearDateFilters 		: BOOL;

eSelectedReportType     : E_ReportType;

iSelectedRow            : INT := 0;
sSelectedPrimaryID      : STRING(50);
sSelectedReportName     : STRING(100);

(***** Search Screen - Datagrid ***********************************************************)

aReportSearchResult     : ARRAY[1..100] OF ST_ReportListItem;
uiReportSearchCount     : UDINT;

(***** Detail Load / PDF Generation *******************************************************)

bLoadSelectedReport     : BOOL;
bLoadBusy               : BOOL;
bLoadDone               : BOOL;
bLoadError              : BOOL;
sLoadStatus             : STRING(100);

bPdfRequest             : BOOL;
bPdfDataReady           : BOOL;
bPdfConsumed            : BOOL;

bListLast100Request 	: BOOL;
bSearchByDateRequest 	: BOOL;
bLoadReportByID 		: BOOL;

(***** Pump Calibration Report Buffers ****************************************************)

// formato generico para tela de pesquisa / selecao
stSelectedCalibReportHeader : ST_CalibrationReportHeader;
aSelectedCalibReportHeader : ARRAY[1..1] OF ST_CalibrationReportHeader;
aSelectedCalibReportLines   : ARRAY[1..300] OF ST_CalibrationReportLine;

// formato compativel com o fluxo atual do relatori.js
aPumpCalibValues        : ARRAY[1..100] OF ST_Data_PCR;

// header copiado campo a campo para casar com o PDF atual
iPumpCalibNo            : DINT;
sPumpCalibUserID        : STRING(50);
sPumpCalibDensity       : STRING(50);
sPumpCalibSolventNo     : STRING(50);
sPumpCalibSolventRev    : STRING(50);
sPumpCalibAllowFail     : STRING(50);
sPumpCalibReplicates    : STRING(50);
sPumpCalibCallInterval  : STRING(50);
sPumpCalibSysRev        : STRING(50);

(***** Method / Recipe Report Buffers *****************************************************)

stMethodHeader          : ST_Parameters_MR;
aMethodVolumeData       : ARRAY[1..10] OF ST_VolumeData;

(***** Complete Method Report Buffers *****************************************************)

aCompleteMethodHeader : ARRAY[1..50] OF ST_CompleteMethodHeader;
aCompleteMethodReport : ARRAY[1..50] OF ST_CompleteMethod;
bBuildCompleteMethodReport : BOOL;

(***** Post Run Report Buffers ************************************************************)

stRunHeader             : ST_PostRunReport;
stRunMethodHeader       : ST_Parameters_MR;
aRunVolumeData          : ARRAY[1..10] OF ST_VolumeData;

(***** System Reports Buffers *************************************************************)

aSelectedSystemSettingsBuf 	: ARRAY[1..1] OF ST_SystemSettingsReport;
stSelectedSystemSettings 	: ST_SystemSettingsReport;
stCurrentSystem         	: ST_SysParameters;
aSystemHistory          	: ARRAY[1..600] OF ST_SysParameters;
bBuildSystemHistoryReport   : BOOL;
sQuickReportName 			: STRING(50);
bBuildLinearHistoryReport   : BOOL;
aLinearHistory           	: ARRAY[1..200] OF ST_LinearReport;

(***** Linear Report Buffers **************************************************************)

stLinearReport 			: ST_LinearReport;

(***** User Reports Buffers ***************************************************************)

aUserHistory            : ARRAY[1..1000] OF ST_Data_CUL;
aCurrentUsers           : ARRAY[1..500] OF ST_Data_CUL;

END_VAR

// ---- GVLs/GVL_Retain.TcGVL
{attribute 'qualified_only'}
VAR_GLOBAL PERSISTENT RETAIN
	
	rValveLastPosition 	: ARRAY[1..5] OF LREAL; //Saves valves position to set the same position on startup [this is because we are using a single turn encoder and a 1:20 ratio gearbox]  
	bPositionIsValid   	: ARRAY[1..5] OF BOOL;  //Position valid flag

	//Counting and stored info for reports and accountability
	iRunNumber : UDINT;
	iCalibrationNumber : UDINT := 0;
	
	(* Calibration *)
	rLinearPumpOldPosition		: ARRAY[1..10] OF LREAL; // Linear pumps old position showed on HMI
	rLinearPumpsLastAdjustUser	: STRING(128);		 	 // Linear pumps last adjusted username
	rLinearPumpsLastAdjustDate	: DATE;				 	 // Linear pumps last adjusted Date
	iPumpCalibrationCount		: UDINT; 				 // Pump Calibration counting number to register on report
	
	aCalibrationPumpFactor		: ARRAY[1..10] OF LREAL := [0.1, 0.1, 0.1, 0.1, 0.1, 0.1, 0.1, 0.1, 0.1, 0.1]; 	 // Pump Factor for rotary pump
	
	(**)
		
END_VAR

// ---- GVLs/GVL_Settings.TcGVL
{attribute 'qualified_only'}
VAR_GLOBAL PERSISTENT
	
	(* System Settings *) //---------------------------------------------------------------------------------------------- 
	sysRevNumber				: INT;
	sLastSysSettingsChangedBy 	: STRING(256);
	sLastSysSettingsChangedOn 	: STRING(256);
	
	stMachineParam				: ST_HMIParameters;						// Motion Parameters to be used on the software
	stCalibParameters 			: ST_CalibrationSettings;				// Calibration Parameters to be used on the software
	stPumpParameters			: ST_PumpSettings;						// Pump Parameters to be used on the software
	stLeakTestParameters		: ST_LeakTestSettings;					// Leak Test Parameters to be used on the software
	stSolventsInfo	 			: ARRAY[1..4] OF ST_SolventsSettings;	// Solvents name and density to be used on the software
	
	bGeneralSealAndPump			: BOOL := FALSE;						// General Settings only parameter SealAndPump
	bDisplayManualControl		: BOOL := FALSE;						// Security Setting parameter Display Manual Control
	bCheckLogonEachRun			: BOOL := FALSE;						// Security Setting parameter Check Logon Each Run
	
	bMeteringSolvent1Done 		: BOOL := FALSE;
	
	(* Scale/Balance comunication *) //-----------------------------------------------------------------------------------
	aBalanceIP		: T_IPv4Addr 	:= '192.168.1.100';	// Scale TCP IP Adress
	nBalancePort	: UINT 			:= 8001;			// TCP port used to communicate with the scale
	
	(* Air Supply Parameters *) //----------------------------------------------------------------------------------------
	rAirSupplyThreshold		: REAL	:= 4.0;
	rAirSupplyTestingTime	: TIME 	:= T#5S;
	
	

END_VAR

// ---- GVLs/GVL_Motion.TcGVL
{attribute 'qualified_only'}
VAR_GLOBAL
	
	M1Motor		: ST_AX8108; //M1 Motor - vertical Axis Stage Collection
	M2Motor		: ST_EL7211; //M2 Motor - vertical Axis Sample Recovery
	M3Motor		: ST_EL7211; //M3 Motor - Horizontal Axis Sample Recovery
	
	aValves		: ARRAY[1..5] OF ST_EP9208;  //M4 to M8 ServoMotor - VICI 6-position Valve 1 to 5
	aPumps		: ARRAY[1..10] OF ST_EL7062; //Pump 1 to 10 StepMotor - Linear and Rotary Actuators
	
	aMotors 	: ARRAY[1..3] OF FB_MotorWrapper; 	//Object Motors Wrapper Instance
	aValvesObj 	: ARRAY[1..5] OF FB_MotorWrapper; 	//Object Motors Wrapper Instance
	aPumpsLinear: ARRAY[1..10] OF FB_MotorWrapper;	//Object Motors Wrapper Instance
	aPumpsRotary: ARRAY[1..10] OF FB_MotorWrapper;	//Object Motors Wrapper Instance
	
	bInitialHomingDone	: BOOL := FALSE; //Flag to check if the initial home was done. Motors homing only happens once when machine is powered up. 
	//bMotorsHomeDone		: BOOL := FALSE;
	
	bValvesPositionRecovered	: BOOL := FALSE; // Flag to indetify if the valves position was recovered when the system is powered up. 
	
	bAnyPumpRunning	: BOOL := FALSE; // Flag to tell when there is at least one pump running 
	
END_VAR

// ---- GVLs/GVL_Recipe.TcGVL
{attribute 'qualified_only'}
VAR_GLOBAL
	
	//Recipe Parameters from HMI
	stInfo			: ST_RecipeInfo;			// info Parameters
	stSolventNTimes	: ST_RecipeSolventAndTimes;	// Solvent and Times Parameters
	stVolumes		: ST_RecipeVolumes;			// Volumes Parameters
	stOtherParams	: ST_RecipeOtherParams;		// Other Parameters
	stFileInfo		: ST_RecipeFileInfo;		// Json file info
	
	stCurrentRecipe : ST_Recipe; // Used by HMI and active cycle
    stActiveRecipe  : ST_Recipe; // Applied in the process
	
	sSelectedRecipeName	: STRING(256); //Json filename 
	
	//aAvailableFiles : ARRAY[0..49] OF ST_RecipeFileInfo; // Recipe folder files
    //iFileCount      : INT;
	
	bIsThereRecipeActivated	: BOOL := FALSE; //Flag to identify if there is a recipe activated before start the autocycle. 	
	
END_VAR

// ---- GVLs/GVL_Safety.TcGVL
{attribute 'qualified_only'}
VAR_GLOBAL
	//Safety All set and enabled to run the machine	
	bSafetyEnable			AT %I* : BOOL;
	bImmediateFaultCommand	AT %Q* : BOOL;
	
	//EL6910 Safety project Variables
	bSafetyErrorAck			AT %Q* : BOOL;
	bSafetyRun				AT %Q* : BOOL;
	bSafetyRestart			AT %Q* : BOOL;
	
	//Motors variables 
	//AX8000 M1 Drive Safety Error Ack and Run
	bM1STOErrorAck			AT %I* : BOOL;
	bSTOErrorAckPulse		AT %I* : BOOL;
	iMotorsSTOEnabled		AT %I* : BOOL;
	
	//AX8000 M4 - M8 Drive Safety Error Ack and Run
	iM4STOErrorAck			AT %Q* : BOOL;
	iM4STORun				AT %Q* : BOOL;
	iM5STOErrorAck			AT %Q* : BOOL;
	iM5STORun				AT %Q* : BOOL;
	iM6STOErrorAck			AT %Q* : BOOL;
	iM6STORun				AT %Q* : BOOL;
	iM7STOErrorAck			AT %Q* : BOOL;
	iM7STORun				AT %Q* : BOOL;
	iM8STOErrorAck			AT %Q* : BOOL;
	iM8STORun				AT %Q* : BOOL;

	//reset button blink signal
	bResetButtonBlink		AT %I*	: BOOL; 
	
	SafetyInputs			AT %I*	: ST_SafetyInputs;
	SafetyOutputs			AT %Q*	: ST_SafetyOutputs;
	
	//STO Monitoring M1 > M8
	bM1STOEnabled			AT %I*	: BOOL;
	bM2STOEnabled			AT %I*	: BOOL;
	bM3STOEnabled			AT %I*	: BOOL;

	//Doors Logic Safety Alias Data exchange
	bDoorClosedAlias		AT %I*	: BOOL;
	bTopDoorsClosedFeedback AT %I*	: BOOL;
	bDoorLockedFeedback		AT %I*	: BOOL;
	bDoorLockCommand		AT %Q*	: BOOL;
	bDoor3BypassAccepted	AT %Q*	: BOOL;
	
	//Air Supply Safety Alias Data exchange
	bAirSupplyEnable		AT %Q*	: BOOL;
	bAirSupplyReset			AT %Q*	: BOOL;
	bAirEnabledFeedback		AT %I* 	: BOOL;
	
	//EL2904 Monitoring Outputs
	aEL2904_T07				AT %I*	: ARRAY[1..4] OF BOOL;
	aEL2904_T08				AT %I*	: ARRAY[1..4] OF BOOL;
	aEL2904_T19				AT %I*	: ARRAY[1..4] OF BOOL;

END_VAR

// ---- GVLs/GVL_UserManagement.TcGVL
{attribute 'qualified_only'}
VAR_GLOBAL
	
	newUser			: STRING;
	newUserGroup	: STRING;
	newUserAutoL	: STRING;
	newUserPassword	: STRING;
	
END_VAR

// ---- POUs/MARCO/DB/GVL_DB.TcGVL
{attribute 'qualified_only'}
{attribute 'TcHmiSymbol' := 'true'}
VAR_GLOBAL
	
	bStartWrite : BOOL;
	bGeneratePDF: BOOL;
	bGeneratePDF2: BOOL;
	bStartRead: BOOL;
	bPreview: BOOL;
	localPDF : STRING;
	testPath : T_MaxString;
	sJsonOutput: STRING(100000);
	stReportHead: ST_ReportInfo;
	
(***** SQL Commands ***********************************************************************************)

//RUN CMDS	
isrtRun: STRING(5000) := 'INSERT INTO [dbo].[RUNS] ( [analyst], [comment], [softwareVersion], [sysMasterRevision], [sysSettingsRevision], [meterVelocity], [runVelocity], [emptyTubesFactor], [fillTubesFactor], [solvent1NameRevision], [solvent2NameRevision], [solvent3NameRevision], [solvent4NameRevision], [timeEventStarted], [timeEventCompleted], [methodID], [CalibrationNo]) VALUES ( $'#1#$', $'#2#$', $'#3#$', $'#4#$', $'#5#$', $'#6#$', $'#7#$', $'#8#$', $'#9#$', $'#10#$', $'#11#$', $'#12#$', $'#13#$', $'#14#$', $'#15#$', #16#, #17#) ';
//slctLastRun: STRING(1000) := 'SELECT TOP 1 [runNo], [analyst], [comment], [softwareVersion], [sysMasterRevision], [sysSettingsRevision], [meterVelocity], [runVelocity], [emptyTubesFactor], [fillTubesFactor], [solvent1NameRevision], [solvent2NameRevision], [solvent3NameRevision], [solvent4NameRevision], [timeEventStarted], [timeEventCompleted], [methodID], [CalibrationNo] FROM [dbo].[RUNS] ORDER BY [runNo] DESC;';

//METHOD CMDS
slctAllMethods: STRING(5000) := 'SELECT [methodName], [methodRevision] FROM [dbo].[METHODS] ';
slctAllActvMethod: STRING(5000) := 'SELECT [methodName], [methodRevision] FROM [dbo].[METHODS] WHERE [methodStatus] = $'activated$'';
slctMethod: STRING(5000) := 'SELECT [methodName], [methodRevision], [methodCreatedBy], [methodCreatedOn], [solvent_R1], [solvent_R2], [solvent_W1], [solvent_W2], [time_R1], [time_R2], [time_W1], [time_W2], [velocity_R1], [velocity_R2], [velocity_W1], [velocity_W2], [soakTime], [agitate_1_Time], [agitate_2_Time], [vialsToFill], [vialPrimeVol], [vial_1_FillVol], [vial_2_4_FillVol], [airDryTime], [methodID], [methodStatus] FROM [dbo].[METHODS] WHERE [methodName] = $'#1#$' AND [methodRevision] = $'#2#$' ';
slctVD: STRING(5000) := 'SELECT [VD_ID], [pump], [stage], [rinse1], [rinse2], [wash1], [wash2], [methodID] FROM [dbo].[VOLUME_DATA] WHERE [methodID] = #1# ';
slctMethodID: STRING(5000) := 'SELECT TOP 1 [methodID] FROM [dbo].[METHODS] WHERE [methodName] = $'#1#$' ORDER BY [methodID] DESC;';
isrtNewMethod: STRING(5000) := 'INSERT INTO [dbo].[METHODS] ( [methodName], [methodRevision], [methodCreatedBy], [methodCreatedOn], [solvent_R1], [solvent_R2], [solvent_W1], [solvent_W2], [time_R1], [time_R2], [time_W1], [time_W2], [velocity_R1], [velocity_R2], [velocity_W1], [velocity_W2], [soakTime], [agitate_1_Time], [agitate_2_Time], [vialsToFill], [vialPrimeVol], [vial_1_FillVol], [vial_2_4_FillVol], [airDryTime], [methodStatus]) VALUES ( $'#1#$', $'#2#$', $'#3#$', $'#4#$', $'#5#$', $'#6#$', $'#7#$', $'#8#$', $'#9#$', $'#10#$', $'#11#$', $'#12#$', $'#13#$', $'#14#$', $'#15#$', $'#16#$', $'#17#$', $'#18#$', $'#19#$', $'#20#$', $'#21#$', $'#22#$', $'#23#$', $'#24#$', $'#25#$') ';
isrtVD: string(5000) := 'INSERT INTO [dbo].[VOLUME_DATA] ( [pump], [stage], [rinse1], [rinse2], [wash1], [wash2], [methodID]) VALUES ( $'#1#$', $'#2#$', $'#3#$', $'#4#$', $'#5#$', $'#6#$', #7#) ';
updtDactvMethod: STRING(5000) := 'UPDATE [dbo].[METHODS] SET [methodStatus] = $'deactivated$' WHERE [methodName] = $'#1#$' AND [methodRevision] = $'#2#$'';

//CALIBRATION CMD
slctLastCalibID: T_Maxstring := 'SELECT TOP 1 [calibrationNo] FROM [dbo].[CALIBRATION_HEAD] ORDER BY [calibrationNo] DESC;';
slctLastCalib: STRING(5000) := 'SELECT TOP 1 [dateTime], [pumpNo], [step], [tareWt], [grossWt], [netVolume], [netWt], [targetVolume], [differencePercent], [criteria], [pumpRevs], [CalibrationNo] FROM [dbo].[CALIBRATION] ORDER BY [calibrationNo] DESC; ';
isrtCalib: STRING(5000) := 'INSERT INTO [dbo].[CALIBRATION_HEAD] ( [userID], [density], [solventNo], [solventRevision], [allowableFail], [replicates], [callInterval], [sysRevisionNo]) VALUES ( $'#1#$', $'#2#$', $'#3#$', $'#4#$', $'#5#$', $'#6#$', $'#7#$', #8#) ';
isrtCalibValues: STRING(5000) := 'INSERT INTO [dbo].[CALIBRATION] ( [dateTime], [pumpNo], [step], [tareWt], [grossWt], [netVolume], [netWt], [targetVolume], [differencePercent], [criteria], [pumpRevs], [CalibrationNo]) VALUES ( $'#1#$', $'#2#$', $'#3#$', $'#4#$', $'#5#$', $'#6#$', $'#7#$', $'#8#$', $'#9#$', $'#10#$', $'#11#$', #12#) ';
dltCalibHead : STRING(500) :='DELETE FROM [dbo].[CALIBRATION_HEAD] WHERE [calibrationNo] = #1#';

//SYSTEM CMD
slctLastSys: STRING(5000) := 'SELECT TOP 1 [gen_SealAndPump], [cal_AcceptanceCriteria], [cal_AllowableFail], [cal_Replicates], [cal_PumpCallIntervalDays], [cal_CloseAppOnCompletation], [AirDryTimeOnCompletation], [lkt_AllowableLeakTestFail], [lkt_LeakTestBuildupTime], [lkt_LeakTestHoldTime], [lkt_LeakTestPressure], [mec_PlatesClosedPosition], [mec_PlatesDryPosition], [mec_PlatesVelocity], [mec_MaxCurrentFastDown], [mec_MaxCurrentSlowDown], [mec_MaxCurrentSlowUp], [pmp_MeterVelocity], [pmp_RunVelocity], [pmp_EmptyFactor], [pmp_FillSolventTubesFactor], [smp_AboveCalibration], [smp_VialSetSpacing], [smp_IntoResBottom], [smp_IntoResDispense], [smp_IntoResWeigh], [smp_IntoVials], [sec_DisplayManualControl], [sec_CheckLogonEachRun], [createdBy], [createdDate], [sysRevisionNo], [smp_AboveVialSet1], [smp_IntoWaste] FROM [dbo].[SYSTEM] ORDER BY [sysRevisionNo] DESC; ';
slctAllSys: STRING(5000) := 'SELECT [gen_SealAndPump], [cal_AcceptanceCriteria], [cal_AllowableFail], [cal_Replicates], [cal_PumpCallIntervalDays], [cal_CloseAppOnCompletation], [AirDryTimeOnCompletation], [lkt_AllowableLeakTestFail], [lkt_LeakTestBuildupTime], [lkt_LeakTestHoldTime], [lkt_LeakTestPressure], [mec_PlatesClosedPosition], [mec_PlatesDryPosition], [mec_PlatesVelocity], [mec_MaxCurrentFastDown], [mec_MaxCurrentSlowDown], [mec_MaxCurrentSlowUp], [pmp_MeterVelocity], [pmp_RunVelocity], [pmp_EmptyFactor], [pmp_FillSolventTubesFactor], [smp_AboveCalibration], [smp_VialSetSpacing], [smp_IntoResBottom], [smp_IntoResDispense], [smp_IntoResWeigh], [smp_IntoVials], [sec_DisplayManualControl], [sec_CheckLogonEachRun], [createdBy], [createdDate], [sysRevisionNo], [smp_AboveVialSet1], [smp_IntoWaste] FROM [dbo].[SYSTEM] ORDER BY [sysRevisionNo] DESC; ';
isrtSys: STRING(5000) := 'INSERT INTO [dbo].[SYSTEM] ( [gen_SealAndPump], [cal_AcceptanceCriteria], [cal_AllowableFail], [cal_Replicates], [cal_PumpCallIntervalDays], [cal_CloseAppOnCompletation], [AirDryTimeOnCompletation], [lkt_AllowableLeakTestFail], [lkt_LeakTestBuildupTime], [lkt_LeakTestHoldTime], [lkt_LeakTestPressure], [mec_PlatesClosedPosition], [mec_PlatesDryPosition], [mec_PlatesVelocity], [mec_MaxCurrentFastDown], [mec_MaxCurrentSlowDown], [mec_MaxCurrentSlowUp], [pmp_MeterVelocity], [pmp_RunVelocity], [pmp_EmptyFactor], [pmp_FillSolventTubesFactor], [smp_AboveCalibration], [smp_VialSetSpacing], [smp_IntoResBottom], [smp_IntoResDispense], [smp_IntoResWeigh], [smp_IntoVials], [sec_DisplayManualControl], [sec_CheckLogonEachRun], [createdBy], [createdDate], [smp_AboveVialSet1], [smp_IntoWaste]) VALUES ( $'#1#$', $'#2#$', $'#3#$', $'#4#$', $'#5#$', $'#6#$', $'#7#$', $'#8#$', $'#9#$', $'#10#$', $'#11#$', $'#12#$', $'#13#$', $'#14#$', $'#15#$', $'#16#$', $'#17#$', $'#18#$', $'#19#$', $'#20#$', $'#21#$', $'#22#$', $'#23#$', $'#24#$', $'#25#$', $'#26#$', $'#27#$', $'#28#$', $'#29#$', $'#30#$', $'#31#$', $'#32#$', $'#33#$') ';

//USERS CMD
isrtUser: STRING(5000) := 'INSERT INTO [dbo].[USERS] ( [userID], [acessLevel], [transactionType], [transactionDate], [transactedBy], [addDate], [enteredBy]) VALUES ( $'#1#$', $'#2#$', $'#3#$', $'#4#$', $'#5#$', $'#6#$', $'#7#$') ';
slctCurrentUser: STRING(5000) := 'SELECT [ID_user], [userID], [acessLevel], [transactionType], [transactionDate], [transactedBy], [addDate], [enteredBy] FROM (SELECT *, ROW_NUMBER() OVER (PARTITION BY [userID] ORDER BY TRY_CONVERT(datetime, [transactionDate], 113) DESC, [ID_user] DESC) AS rn FROM [dbo].[USERS] WHERE [transactionType] = $'Added$') t WHERE rn = 1 AND NOT EXISTS (SELECT 1 FROM [dbo].[USERS] r WHERE r.[userID] = t.[userID] AND r.[transactionType] = $'Removed$' AND TRY_CONVERT(datetime, r.[transactionDate], 113) > TRY_CONVERT(datetime, t.[transactionDate], 113));';
slctAllUsers: STRING(5000) := 'SELECT [ID_user], [userID], [acessLevel], [transactionType], [transactionDate], [transactedBy], [addDate], [enteredBy] FROM [dbo].[USERS] ';

//SOLVENTS
isrtSolvent: STRING(1000) := 'INSERT INTO [dbo].[SOLVENTS] ( [solventName1], [solventName2], [solventName3], [solventName4], [density1], [density2], [density3], [density4], [addedBy], [addedDate]) VALUES ( $'#1#$', $'#2#$', $'#3#$', $'#4#$', $'#5#$', $'#6#$', $'#7#$', $'#8#$', $'#9#$', $'#10#$') ';
slctSolvent: STRING(1000) := 'SELECT TOP 1 [SOLVENT_ID], [solventName1], [solventName2], [solventName3], [solventName4], [density1], [density2], [density3], [density4], [addedBy], [addedDate] FROM [dbo].[SOLVENTS] ORDER BY [SOLVENT_ID] DESC; ';
slctAllSolvents: STRING(1000) := 'SELECT [SOLVENT_ID], [solventName1], [solventName2], [solventName3], [solventName4], [density1], [density2], [density3], [density4], [addedBy], [addedDate] FROM [dbo].[SOLVENTS] ';

//LINEAR MOTORS
isrtLinear: STRING(1500) := 'INSERT INTO [dbo].[LINEAR] ( [pump1], [pump2], [pump3], [pump4], [pump5], [pump6], [pump7], [pump8], [pump9], [pump10], [changedBy], [changedOn]) VALUES ( $'#1#$', $'#2#$', $'#3#$', $'#4#$', $'#5#$', $'#6#$', $'#7#$', $'#8#$', $'#9#$', $'#10#$', $'#11#$', $'#12#$') ';
slctLinear: STRING(1000) := 'SELECT TOP 1 [ID_Linear], [pump1], [pump2], [pump3], [pump4], [pump5], [pump6], [pump7], [pump8], [pump9], [pump10] FROM [dbo].[LINEAR] ORDER BY [ID_Linear] DESC; ';

//PUMP CALIBRATION REPORT / HISTORY CMD
slctCalibReportList: STRING(5000) := 'SELECT TOP 50 [CalibrationNo], [userID], [solventNo], [sysRevisionNo] FROM [dbo].[PumpCalibrationHeader] ORDER BY [CalibrationNo] DESC;';
slctPumpCalibHeaderByNo: STRING(5000) := 'SELECT TOP 1 [CalibrationNo], [userID], [density], [solventNo], [solventRevision], [allowableFail], [replicates], [callInterval], [sysRevisionNo] FROM [dbo].[PumpCalibrationHeader] WHERE [CalibrationNo] = #1#;';
slctPumpCalibValuesByNo: STRING(5000) := 'SELECT [CalibrationNo], [dateTime], [pumpNo], [step], [tareWt], [grossWt], [netVolume], [netWt], [targetVolume], [differencePercent], [criteria], [pumpRevs] FROM [dbo].[PumpCalibrationValues] WHERE [CalibrationNo] = #1# ORDER BY [ID] ASC;';

slctCalibReportListFromValues: STRING(5000) := 'SELECT TOP 100 CAST(ISNULL([ReportType], $'$') AS VARCHAR(50)) AS [ReportType], CAST(ISNULL([ReportID], $'$') AS VARCHAR(50)) AS [ReportID], CAST(ISNULL([CreatedOn], $'$') AS VARCHAR(30)) AS [CreatedOn], CAST(ISNULL([CreatedBy], $'$') AS VARCHAR(50)) AS [CreatedBy], CAST(ISNULL([Description], $'$') AS VARCHAR(200)) AS [Description], CAST(ISNULL([sPrimaryKey], $'$') AS VARCHAR(50)) AS [sPrimaryKey] FROM [dbo].[vw_ReportList_PumpCalibration] ORDER BY CAST([ReportID] AS INT) DESC;';
slctMethodReportList: STRING(5000) := 'SELECT TOP 50 $'Method$' AS [ReportType], CAST([methodID] AS VARCHAR(50)) AS [ReportID], [methodCreatedOn] AS [CreatedOn], [methodCreatedBy] AS [CreatedBy], [methodName] + $' Rev $' + [methodRevision] AS [Description], CAST([methodID] AS VARCHAR(50)) AS [sPrimaryKey] FROM [dbo].[METHODS] ORDER BY [methodID] DESC;';
slctRunReportList: STRING(5000) := 'SELECT TOP 100 CAST(ISNULL($'Run$', $'$') AS VARCHAR(50)) AS [ReportType], CAST(ISNULL(CAST([runNo] AS VARCHAR(50)), $'$') AS VARCHAR(50)) AS [ReportID], CAST(ISNULL([timeEventCompleted], $'$') AS VARCHAR(30)) AS [CreatedOn], CAST(ISNULL([analyst], $'$') AS VARCHAR(50)) AS [CreatedBy], CAST(ISNULL($'Method ID $' + CAST([methodID] AS VARCHAR(20)) + $' / Cal $' + CAST([CalibrationNo] AS VARCHAR(20)) + CASE WHEN ISNULL([comment], $'$') = $'$' THEN $'$' ELSE $' - $' + [comment] END, $'$') AS VARCHAR(200)) AS [Description], CAST(ISNULL(CAST([runNo] AS VARCHAR(50)), $'$') AS VARCHAR(50)) AS [sPrimaryKey] FROM [dbo].[RUNS] ORDER BY [runNo] DESC;';
slctLinearReportList: STRING(5000) := 'SELECT TOP 50 $'Linear$' AS [ReportType], CAST([ID_Linear] AS VARCHAR(50)) AS [ReportID], $'$' AS [CreatedOn], $'$' AS [CreatedBy], $'Linear pump positions set $' + CAST([ID_Linear] AS VARCHAR(20)) AS [Description], CAST([ID_Linear] AS VARCHAR(50)) AS [sPrimaryKey] FROM [dbo].[LINEAR] ORDER BY [ID_Linear] DESC;';

// REPORT SCREEN LISTING AND SELECTING
slctPumpCalibHeaderByNo1: STRING(5000) := 'SELECT TOP 1 CAST($'Pump Calibration$' AS VARCHAR(50)) AS [sReportId], CAST(ISNULL([CalibrationNo], $'$') AS VARCHAR(30)) AS [sCalibrationNo], CAST(ISNULL([userID], $'$') AS VARCHAR(50)) AS [sUserId], CAST(ISNULL([density], $'$') AS VARCHAR(30)) AS [sDensity], CAST(ISNULL([solventNo], $'$') AS VARCHAR(30)) AS [sSolventNo], CAST(ISNULL([solventRevision], $'$') AS VARCHAR(30)) AS [sSolventRevision], CAST(ISNULL([sysRevisionNo], $'$') AS VARCHAR(30)) AS [sSysRevisionNo], CAST(ISNULL([allowableFail], $'$') AS VARCHAR(30)) AS [sAllowableFail], CAST(ISNULL([replicates], $'$') AS VARCHAR(30)) AS [sReplicates], CAST(ISNULL([callInterval], $'$') AS VARCHAR(30)) AS [sCallInterval], CAST($'$' AS VARCHAR(30)) AS [sCreatedAt] FROM [dbo].[CALIBRATION_HEAD] WHERE [CalibrationNo] = #1#;';
slctPumpCalibValuesByNo1: STRING(5000) := 'SELECT CAST(ISNULL([dateTime], $'$') AS VARCHAR(40)) AS [sDateTime], CAST(ISNULL([pumpNo], $'$') AS VARCHAR(10)) AS [sPumpNo], CAST(ISNULL([step], $'$') AS VARCHAR(20)) AS [sStep], CAST(ISNULL([tareWt], $'$') AS VARCHAR(30)) AS [sTareWt], CAST(ISNULL([grossWt], $'$') AS VARCHAR(30)) AS [sGrossWt], CAST(ISNULL([netWt], $'$') AS VARCHAR(30)) AS [sNetWt], CAST(ISNULL([netVolume], $'$') AS VARCHAR(30)) AS [sNetVolume], CAST(ISNULL([targetVolume], $'$') AS VARCHAR(30)) AS [sTargetVolume], CAST(ISNULL([differencePercent], $'$') AS VARCHAR(30)) AS [sDifferencePercent], CAST(ISNULL([criteria], $'$') AS VARCHAR(20)) AS [sCriteria], CAST(ISNULL([pumpRevs], $'$') AS VARCHAR(30)) AS [sPumpRevs] FROM [dbo].[CALIBRATION] WHERE [CalibrationNo] = #1# ORDER BY [Data_ID] ASC;';
slctSystemSettingsReportList: STRING(5000) := 'SELECT TOP 100 CAST([ReportType] AS VARCHAR(50)) AS [ReportType], CAST([ReportID] AS VARCHAR(50)) AS [ReportID], CAST([CreatedOn] AS VARCHAR(30)) AS [CreatedOn], CAST([CreatedBy] AS VARCHAR(50)) AS [CreatedBy], CAST([Description] AS VARCHAR(200)) AS [Description], CAST([sPrimaryKey] AS VARCHAR(50)) AS [sPrimaryKey] FROM [dbo].[vw_ReportList_SystemSettings] ORDER BY CAST([ReportID] AS INT) DESC;';
slctSystemSettingsByRevision: STRING(5000) := 'SELECT TOP 1 CAST([gen_SealAndPump] AS VARCHAR(100)) AS [sGenSealAndPump], CAST([cal_AcceptanceCriteria] AS VARCHAR(100)) AS [sCalAcceptanceCriteria], CAST([cal_AllowableFail] AS VARCHAR(100)) AS [sCalAllowableFail], CAST([cal_Replicates] AS VARCHAR(100)) AS [sCalReplicates], CAST([cal_PumpCallIntervalDays] AS VARCHAR(100)) AS [sCalPumpCallIntervalDays], CAST([cal_CloseAppOnCompletation] AS VARCHAR(100)) AS [sCalCloseAppOnCompletion], CAST([AirDryTimeOnCompletation] AS VARCHAR(100)) AS [sAirDryTimeOnCompletion], CAST([lkt_AllowableLeakTestFail] AS VARCHAR(100)) AS [sLktAllowableLeakTestFail], CAST([lkt_LeakTestBuildupTime] AS VARCHAR(100)) AS [sLktLeakTestBuildUpTime], CAST([lkt_LeakTestHoldTime] AS VARCHAR(100)) AS [sLktLeakTestHoldTime], CAST([lkt_LeakTestPressure] AS VARCHAR(100)) AS [sLktLeakTestPressure], CAST([mec_PlatesClosedPosition] AS VARCHAR(100)) AS [sMecPlatesClosedPosition], CAST([mec_PlatesDryPosition] AS VARCHAR(100)) AS [sMecPlatesDryPosition], CAST([mec_PlatesVelocity] AS VARCHAR(100)) AS [sMecPlatesVelocity], CAST([mec_MaxCurrentFastDown] AS VARCHAR(100)) AS [sMecMaxCurrentFastDown], CAST([mec_MaxCurrentSlowDown] AS VARCHAR(100)) AS [sMecMaxCurrentSlowDown], CAST([mec_MaxCurrentSlowUp] AS VARCHAR(100)) AS [sMecMaxCurrentSlowUp], CAST([pmp_MeterVelocity] AS VARCHAR(100)) AS [sPmpMeterVelocity], CAST([pmp_RunVelocity] AS VARCHAR(100)) AS [sPmpRunVelocity], CAST([pmp_EmptyFactor] AS VARCHAR(100)) AS [sPmpEmptyFactor], CAST([pmp_FillSolventTubesFactor] AS VARCHAR(100)) AS [sPmpFillSolventTubesFactor], CAST([smp_AboveCalibration] AS VARCHAR(100)) AS [sSmpAboveCalibration], CAST([smp_VialSetSpacing] AS VARCHAR(100)) AS [sSmpVialSetSpacing], CAST([smp_IntoResBottom] AS VARCHAR(100)) AS [sSmpIntoResBottom], CAST([smp_IntoResDispense] AS VARCHAR(100)) AS [sSmpIntoResDispense], CAST([smp_IntoResWeigh] AS VARCHAR(100)) AS [sSmpIntoResWeigh], CAST([smp_IntoVials] AS VARCHAR(100)) AS [sSmpIntoVials], CAST([smp_IntoWaste] AS VARCHAR(100)) AS [sSmpIntoWaste], CAST([sec_DisplayManualControl] AS VARCHAR(100)) AS [sSecDisplayManualControl], CAST([sec_CheckLogonEachRun] AS VARCHAR(100)) AS [sSecCheckLogonEachRun], CAST([createdBy] AS VARCHAR(100)) AS [sCreatedBy], CAST([createdDate] AS VARCHAR(100)) AS [sCreatedDate], CAST([sysRevisionNo] AS VARCHAR(30)) AS [sSysRevisionNo] FROM [dbo].[SYSTEM] WHERE [sysRevisionNo] = #1#;';
slctMethodReportSearchLatest : STRING(5000) := 'SELECT TOP 100 CAST(ISNULL([ReportType], $'$') AS VARCHAR(50)) AS [ReportType], CAST(ISNULL([ReportID], $'$') AS VARCHAR(50)) AS [ReportID], CAST(ISNULL([CreatedOn], $'$') AS VARCHAR(30)) AS [CreatedOn], CAST(ISNULL([CreatedBy], $'$') AS VARCHAR(50)) AS [CreatedBy], CAST(ISNULL([Description], $'$') AS VARCHAR(200)) AS [Description], CAST(ISNULL([sPrimaryKey], $'$') AS VARCHAR(50)) AS [sPrimaryKey] FROM [dbo].[vw_ReportList_Recipe] ORDER BY CAST([ReportID] AS INT) DESC;';
slctMethodHeaderByID : STRING(5000) := 'SELECT TOP 1 CAST(ISNULL([methodName], $'$') AS VARCHAR(100)) AS [methodName], CAST(ISNULL([methodRevision], $'$') AS VARCHAR(100)) AS [methodRevision], CAST(ISNULL([methodCreatedBy], $'$') AS VARCHAR(100)) AS [methodCreatedBy], CAST(ISNULL([methodCreatedOn], $'$') AS VARCHAR(100)) AS [methodCreatedOn], CAST(ISNULL([solvent_R1], $'$') AS VARCHAR(100)) AS [solvent_R1], CAST(ISNULL([solvent_R2], $'$') AS VARCHAR(100)) AS [solvent_R2], CAST(ISNULL([solvent_W1], $'$') AS VARCHAR(100)) AS [solvent_W1], CAST(ISNULL([solvent_W2], $'$') AS VARCHAR(100)) AS [solvent_W2], CAST(ISNULL([time_R1], $'$') AS VARCHAR(100)) AS [time_R1], CAST(ISNULL([time_R2], $'$') AS VARCHAR(100)) AS [time_R2], CAST(ISNULL([time_W1], $'$') AS VARCHAR(100)) AS [time_W1], CAST(ISNULL([time_W2], $'$') AS VARCHAR(100)) AS [time_W2], CAST(ISNULL([velocity_R1], $'$') AS VARCHAR(100)) AS [velocity_R1], CAST(ISNULL([velocity_R2], $'$') AS VARCHAR(100)) AS [velocity_R2], CAST(ISNULL([velocity_W1], $'$') AS VARCHAR(100)) AS [velocity_W1], CAST(ISNULL([velocity_W2], $'$') AS VARCHAR(100)) AS [velocity_W2], CAST(ISNULL([soakTime], $'$') AS VARCHAR(100)) AS [soakTime], CAST(ISNULL([agitate_1_Time], $'$') AS VARCHAR(100)) AS [agitate_1_Time], CAST(ISNULL([agitate_2_Time], $'$') AS VARCHAR(100)) AS [agitate_2_Time], CAST(ISNULL([vialsToFill], $'$') AS VARCHAR(100)) AS [vialsToFill], CAST(ISNULL([vialPrimeVol], $'$') AS VARCHAR(100)) AS [vialPrimeVol], CAST(ISNULL([vial_1_FillVol], $'$') AS VARCHAR(100)) AS [vial_1_FillVol], CAST(ISNULL([vial_2_4_FillVol], $'$') AS VARCHAR(100)) AS [vial_2_4_FillVol], CAST(ISNULL([airDryTime], $'$') AS VARCHAR(100)) AS [airDryTime], ISNULL([methodID], 0) AS [methodID], CAST(ISNULL([methodStatus], $'$') AS VARCHAR(100)) AS [methodStatus] FROM [dbo].[METHODS] WHERE [methodID] = #1#;';
slctMethodVolumeByID : STRING(5000) := 'SELECT ISNULL([VD_ID], 0) AS [VD_ID], CAST(ISNULL([pump], $'$') AS VARCHAR(100)) AS [pump], CAST(ISNULL([stage], $'$') AS VARCHAR(100)) AS [stage], CAST(ISNULL([rinse1], $'$') AS VARCHAR(100)) AS [rinse1], CAST(ISNULL([rinse2], $'$') AS VARCHAR(100)) AS [rinse2], CAST(ISNULL([wash1], $'$') AS VARCHAR(100)) AS [wash1], CAST(ISNULL([wash2], $'$') AS VARCHAR(100)) AS [wash2], ISNULL([methodID], 0) AS [methodID] FROM [dbo].[VOLUME_DATA] WHERE [methodID] = #1# ORDER BY [VD_ID] ASC;';
slctPostRunHeaderByID : STRING(5000) := 'SELECT TOP 1 ISNULL([runNo], 0) AS [runNo], CAST(ISNULL([analyst], $'$') AS VARCHAR(100)) AS [analyst], CAST(ISNULL([comment], $'$') AS VARCHAR(100)) AS [comment], CAST(ISNULL([softwareVersion], $'$') AS VARCHAR(100)) AS [softwareVersion], CAST(ISNULL([sysMasterRevision], $'$') AS VARCHAR(100)) AS [sysMasterRevision], CAST(ISNULL([sysSettingsRevision], $'$') AS VARCHAR(100)) AS [sysSettingsRevision], CAST(ISNULL([meterVelocity], $'$') AS VARCHAR(100)) AS [meterVelocity], CAST(ISNULL([runVelocity], $'$') AS VARCHAR(100)) AS [runVelocity], CAST(ISNULL([emptyTubesFactor], $'$') AS VARCHAR(100)) AS [emptyTubesFactor], CAST(ISNULL([fillTubesFactor], $'$') AS VARCHAR(100)) AS [fillTubesFactor], CAST(ISNULL([solvent1NameRevision], $'$') AS VARCHAR(100)) AS [solvent1NameRevision], CAST(ISNULL([solvent2NameRevision], $'$') AS VARCHAR(100)) AS [solvent2NameRevision], CAST(ISNULL([solvent3NameRevision], $'$') AS VARCHAR(100)) AS [solvent3NameRevision], CAST(ISNULL([solvent4NameRevision], $'$') AS VARCHAR(100)) AS [solvent4NameRevision], CAST(ISNULL([timeEventStarted], $'$') AS VARCHAR(100)) AS [timeEventStarted], CAST(ISNULL([timeEventCompleted], $'$') AS VARCHAR(100)) AS [timeEventCompleted], ISNULL([methodID], 0) AS [methodID], ISNULL([CalibrationNo], 0) AS [CalibrationNo] FROM [dbo].[RUNS] WHERE [runNo] = #1#;';
slctPostRunMethodHeaderByID : STRING(5000) := 'SELECT TOP 1 CAST(ISNULL([methodName], $'$') AS VARCHAR(100)) AS [methodName], CAST(ISNULL([methodRevision], $'$') AS VARCHAR(100)) AS [methodRevision], CAST(ISNULL([methodCreatedBy], $'$') AS VARCHAR(100)) AS [methodCreatedBy], CAST(ISNULL([methodCreatedOn], $'$') AS VARCHAR(100)) AS [methodCreatedOn], CAST(ISNULL([solvent_R1], $'$') AS VARCHAR(100)) AS [solvent_R1], CAST(ISNULL([solvent_R2], $'$') AS VARCHAR(100)) AS [solvent_R2], CAST(ISNULL([solvent_W1], $'$') AS VARCHAR(100)) AS [solvent_W1], CAST(ISNULL([solvent_W2], $'$') AS VARCHAR(100)) AS [solvent_W2], CAST(ISNULL([time_R1], $'$') AS VARCHAR(100)) AS [time_R1], CAST(ISNULL([time_R2], $'$') AS VARCHAR(100)) AS [time_R2], CAST(ISNULL([time_W1], $'$') AS VARCHAR(100)) AS [time_W1], CAST(ISNULL([time_W2], $'$') AS VARCHAR(100)) AS [time_W2], CAST(ISNULL([velocity_R1], $'$') AS VARCHAR(100)) AS [velocity_R1], CAST(ISNULL([velocity_R2], $'$') AS VARCHAR(100)) AS [velocity_R2], CAST(ISNULL([velocity_W1], $'$') AS VARCHAR(100)) AS [velocity_W1], CAST(ISNULL([velocity_W2], $'$') AS VARCHAR(100)) AS [velocity_W2], CAST(ISNULL([soakTime], $'$') AS VARCHAR(100)) AS [soakTime], CAST(ISNULL([agitate_1_Time], $'$') AS VARCHAR(100)) AS [agitate_1_Time], CAST(ISNULL([agitate_2_Time], $'$') AS VARCHAR(100)) AS [agitate_2_Time], CAST(ISNULL([vialsToFill], $'$') AS VARCHAR(100)) AS [vialsToFill], CAST(ISNULL([vialPrimeVol], $'$') AS VARCHAR(100)) AS [vialPrimeVol], CAST(ISNULL([vial_1_FillVol], $'$') AS VARCHAR(100)) AS [vial_1_FillVol], CAST(ISNULL([vial_2_4_FillVol], $'$') AS VARCHAR(100)) AS [vial_2_4_FillVol], CAST(ISNULL([airDryTime], $'$') AS VARCHAR(100)) AS [airDryTime], ISNULL([methodID], 0) AS [methodID], CAST(ISNULL([methodStatus], $'$') AS VARCHAR(100)) AS [methodStatus] FROM [dbo].[METHODS] WHERE [methodID] = #1#;';
slctPostRunVolumeByMethodID : STRING(5000) := 'SELECT ISNULL([VD_ID], 0) AS [VD_ID], CAST(ISNULL([pump], $'$') AS VARCHAR(100)) AS [pump], CAST(ISNULL([stage], $'$') AS VARCHAR(100)) AS [stage], CAST(ISNULL([rinse1], $'$') AS VARCHAR(100)) AS [rinse1], CAST(ISNULL([rinse2], $'$') AS VARCHAR(100)) AS [rinse2], CAST(ISNULL([wash1], $'$') AS VARCHAR(100)) AS [wash1], CAST(ISNULL([wash2], $'$') AS VARCHAR(100)) AS [wash2], ISNULL([methodID], 0) AS [methodID] FROM [dbo].[VOLUME_DATA] WHERE [methodID] = #1# ORDER BY [VD_ID] ASC;';
slctLinearReportSearch : STRING(5000) := 'SELECT TOP 100 CAST(ISNULL([ReportType], $'$') AS VARCHAR(50)) AS [ReportType], CAST(ISNULL([ReportID], $'$') AS VARCHAR(50)) AS [ReportID], CAST(ISNULL([CreatedOn], $'$') AS VARCHAR(30)) AS [CreatedOn], CAST(ISNULL([CreatedBy], $'$') AS VARCHAR(50)) AS [CreatedBy], CAST(ISNULL([Description], $'$') AS VARCHAR(200)) AS [Description], CAST(ISNULL([sPrimaryKey], $'$') AS VARCHAR(50)) AS [sPrimaryKey] FROM [dbo].[vw_ReportList_Linear] ORDER BY CAST([ReportID] AS INT) DESC;';
slctLinearByID : STRING(5000) := 'SELECT TOP 1 ISNULL([ID_Linear], 0) AS [ID_Linear], CAST(ISNULL([pump1], $'$') AS VARCHAR(100)) AS [pump1], CAST(ISNULL([pump2], $'$') AS VARCHAR(100)) AS [pump2], CAST(ISNULL([pump3], $'$') AS VARCHAR(100)) AS [pump3], CAST(ISNULL([pump4], $'$') AS VARCHAR(100)) AS [pump4], CAST(ISNULL([pump5], $'$') AS VARCHAR(100)) AS [pump5], CAST(ISNULL([pump6], $'$') AS VARCHAR(100)) AS [pump6], CAST(ISNULL([pump7], $'$') AS VARCHAR(100)) AS [pump7], CAST(ISNULL([pump8], $'$') AS VARCHAR(100)) AS [pump8], CAST(ISNULL([pump9], $'$') AS VARCHAR(100)) AS [pump9], CAST(ISNULL([pump10], $'$') AS VARCHAR(100)) AS [pump10], CAST(ISNULL([changedBy], $'$') AS VARCHAR(100)) AS [changedBy], CAST(ISNULL([changedOn], $'$') AS VARCHAR(100)) AS [changedOn] FROM [dbo].[LINEAR] WHERE [ID_Linear] = #1#;';
//slctAllMethodsForCompleteReport : STRING(5000) := 'SELECT CAST(ISNULL([methodName], $'$') AS VARCHAR(100)) AS [methodName], CAST(ISNULL([methodRevision], $'$') AS VARCHAR(100)) AS [methodRevision], CAST(ISNULL([methodCreatedBy], $'$') AS VARCHAR(100)) AS [methodCreatedBy], CAST(ISNULL([methodCreatedOn], $'$') AS VARCHAR(100)) AS [methodCreatedOn], CAST(ISNULL([solvent_R1], $'$') AS VARCHAR(100)) AS [solvent_R1], CAST(ISNULL([solvent_R2], $'$') AS VARCHAR(100)) AS [solvent_R2], CAST(ISNULL([solvent_W1], $'$') AS VARCHAR(100)) AS [solvent_W1], CAST(ISNULL([solvent_W2], $'$') AS VARCHAR(100)) AS [solvent_W2], CAST(ISNULL([time_R1], $'$') AS VARCHAR(100)) AS [time_R1], CAST(ISNULL([time_R2], $'$') AS VARCHAR(100)) AS [time_R2], CAST(ISNULL([time_W1], $'$') AS VARCHAR(100)) AS [time_W1], CAST(ISNULL([time_W2], $'$') AS VARCHAR(100)) AS [time_W2], CAST(ISNULL([velocity_R1], $'$') AS VARCHAR(100)) AS [velocity_R1], CAST(ISNULL([velocity_R2], $'$') AS VARCHAR(100)) AS [velocity_R2], CAST(ISNULL([velocity_W1], $'$') AS VARCHAR(100)) AS [velocity_W1], CAST(ISNULL([velocity_W2], $'$') AS VARCHAR(100)) AS [velocity_W2], CAST(ISNULL([soakTime], $'$') AS VARCHAR(100)) AS [soakTime], CAST(ISNULL([agitate_1_Time], $'$') AS VARCHAR(100)) AS [agitate_1_Time], CAST(ISNULL([agitate_2_Time], $'$') AS VARCHAR(100)) AS [agitate_2_Time], CAST(ISNULL([vialsToFill], $'$') AS VARCHAR(100)) AS [vialsToFill], CAST(ISNULL([vialPrimeVol], $'$') AS VARCHAR(100)) AS [vialPrimeVol], CAST(ISNULL([vial_1_FillVol], $'$') AS VARCHAR(100)) AS [vial_1_FillVol], CAST(ISNULL([vial_2_4_FillVol], $'$') AS VARCHAR(100)) AS [vial_2_4_FillVol], CAST(ISNULL([airDryTime], $'$') AS VARCHAR(100)) AS [airDryTime], ISNULL([methodID], 0) AS [methodID], CAST(ISNULL([methodStatus], $'$') AS VARCHAR(100)) AS [methodStatus] FROM [dbo].[METHODS] ORDER BY TRY_CAST([methodID] AS INT) DESC;';
slctAllMethodsForCompleteReport : STRING(5000) := 'SELECT TOP 100 CAST(ISNULL([methodName], $'$') AS VARCHAR(100)) AS [methodName], CAST(ISNULL([methodRevision], $'$') AS VARCHAR(100)) AS [methodRevision], CAST(ISNULL([methodCreatedBy], $'$') AS VARCHAR(100)) AS [methodCreatedBy], CAST(ISNULL([methodCreatedOn], $'$') AS VARCHAR(100)) AS [methodCreatedOn], CAST(ISNULL([solvent_R1], $'$') AS VARCHAR(100)) AS [solvent_R1], CAST(ISNULL([solvent_R2], $'$') AS VARCHAR(100)) AS [solvent_R2], CAST(ISNULL([solvent_W1], $'$') AS VARCHAR(100)) AS [solvent_W1], CAST(ISNULL([solvent_W2], $'$') AS VARCHAR(100)) AS [solvent_W2], CAST(ISNULL([time_R1], $'$') AS VARCHAR(100)) AS [time_R1], CAST(ISNULL([time_R2], $'$') AS VARCHAR(100)) AS [time_R2], CAST(ISNULL([time_W1], $'$') AS VARCHAR(100)) AS [time_W1], CAST(ISNULL([time_W2], $'$') AS VARCHAR(100)) AS [time_W2], CAST(ISNULL([velocity_R1], $'$') AS VARCHAR(100)) AS [velocity_R1], CAST(ISNULL([velocity_R2], $'$') AS VARCHAR(100)) AS [velocity_R2], CAST(ISNULL([velocity_W1], $'$') AS VARCHAR(100)) AS [velocity_W1], CAST(ISNULL([velocity_W2], $'$') AS VARCHAR(100)) AS [velocity_W2], CAST(ISNULL([soakTime], $'$') AS VARCHAR(100)) AS [soakTime], CAST(ISNULL([agitate_1_Time], $'$') AS VARCHAR(100)) AS [agitate_1_Time], CAST(ISNULL([agitate_2_Time], $'$') AS VARCHAR(100)) AS [agitate_2_Time], CAST(ISNULL([vialsToFill], $'$') AS VARCHAR(100)) AS [vialsToFill], CAST(ISNULL([vialPrimeVol], $'$') AS VARCHAR(100)) AS [vialPrimeVol], CAST(ISNULL([vial_1_FillVol], $'$') AS VARCHAR(100)) AS [vial_1_FillVol], CAST(ISNULL([vial_2_4_FillVol], $'$') AS VARCHAR(100)) AS [vial_2_4_FillVol], CAST(ISNULL([airDryTime], $'$') AS VARCHAR(100)) AS [airDryTime], ISNULL([methodID], 0) AS [methodID], CAST(ISNULL([methodStatus], $'$') AS VARCHAR(100)) AS [methodStatus] FROM [dbo].[METHODS] ORDER BY [methodID] DESC;';

// USER MANAGEMENT
//insUserMgmtHistory : STRING(5000) := 'INSERT INTO dbo.UserManagementHistory (TargetUser, EventType, OldGroup, NewGroup, OldAutoLogoutMin, NewAutoLogoutMin, PerformedBy, SourceScreen, EventComment) VALUES ($'#1#$', $'#2#$', $'#3#$', $'#4#$', #5#, #6#, $'#7#$', $'#8#$', $'#9#$');';
slctUserMgmtHistoryList : STRING(5000) := 'SELECT TOP 100 CAST(ISNULL([ID], 0) AS VARCHAR(20)) AS [ID], CAST(ISNULL([EventDate], $'$') AS VARCHAR(30)) AS [EventDate], CAST(ISNULL([TargetUser], $'$') AS VARCHAR(100)) AS [TargetUser], CAST(ISNULL([EventType], $'$') AS VARCHAR(50)) AS [EventType], CAST(ISNULL([OldGroup], $'$') AS VARCHAR(100)) AS [OldGroup], CAST(ISNULL([NewGroup], $'$') AS VARCHAR(100)) AS [NewGroup], CAST(ISNULL([OldAutoLogoutMin], 0) AS VARCHAR(20)) AS [OldAutoLogoutMin], CAST(ISNULL([NewAutoLogoutMin], 0) AS VARCHAR(20)) AS [NewAutoLogoutMin], CAST(ISNULL([PerformedBy], $'$') AS VARCHAR(100)) AS [PerformedBy], CAST(ISNULL([SourceScreen], $'$') AS VARCHAR(100)) AS [SourceScreen], CAST(ISNULL([EventComment], $'$') AS VARCHAR(255)) AS [EventComment] FROM [dbo].[UserManagementHistory] ORDER BY [ID] DESC;';
slctUserMgmtHistoryListByDate : STRING(5000) := 'SELECT TOP 100 CAST(ISNULL([ID], 0) AS VARCHAR(20)) AS [ID], CAST(ISNULL([EventDate], $'$') AS VARCHAR(30)) AS [EventDate], CAST(ISNULL([TargetUser], $'$') AS VARCHAR(100)) AS [TargetUser], CAST(ISNULL([EventType], $'$') AS VARCHAR(50)) AS [EventType], CAST(ISNULL([OldGroup], $'$') AS VARCHAR(100)) AS [OldGroup], CAST(ISNULL([NewGroup], $'$') AS VARCHAR(100)) AS [NewGroup], CAST(ISNULL([OldAutoLogoutMin], 0) AS VARCHAR(20)) AS [OldAutoLogoutMin], CAST(ISNULL([NewAutoLogoutMin], 0) AS VARCHAR(20)) AS [NewAutoLogoutMin], CAST(ISNULL([PerformedBy], $'$') AS VARCHAR(100)) AS [PerformedBy], CAST(ISNULL([SourceScreen], $'$') AS VARCHAR(100)) AS [SourceScreen], CAST(ISNULL([EventComment], $'$') AS VARCHAR(255)) AS [EventComment] FROM [dbo].[UserManagementHistory] WHERE [EventDate] >= #1# AND [EventDate] <= #2# ORDER BY [EventDate] DESC, [ID] DESC;';
//slctUserMgmtHistoryByUser : STRING(5000) := 'SELECT TOP 100 CAST(ISNULL([ID], 0) AS VARCHAR(20)) AS [ID], CAST(ISNULL([EventDate], $'$') AS VARCHAR(30)) AS [EventDate], CAST(ISNULL([TargetUser], $'$') AS VARCHAR(100)) AS [TargetUser], ' +'CAST(ISNULL([EventType], $'$') AS VARCHAR(50)) AS [EventType], CAST(ISNULL([OldGroup], $'$') AS VARCHAR(100)) AS [OldGroup], CAST(ISNULL([NewGroup], $'$') AS VARCHAR(100)) AS [NewGroup], CAST(ISNULL([OldAutoLogoutMin], 0) AS VARCHAR(20)) AS [OldAutoLogoutMin], CAST(ISNULL([NewAutoLogoutMin], 0) AS VARCHAR(20)) AS [NewAutoLogoutMin], CAST(ISNULL([PerformedBy], $'$') AS VARCHAR(100)) AS [PerformedBy], CAST(ISNULL([SourceScreen], $'$') AS VARCHAR(100)) AS [SourceScreen], CAST(ISNULL([EventComment], $'$') AS VARCHAR(255)) AS [EventComment] FROM [dbo].[UserManagementHistory] WHERE [TargetUser] = $'#1#$' ORDER BY [ID] DESC;';
isrtUserMgmtHistory : STRING(5000) := 'INSERT INTO dbo.UserManagementHistory (TargetUser, EventType, OldGroup, NewGroup, OldAutoLogoutMin, NewAutoLogoutMin, PerformedBy, SourceScreen, EventComment) VALUES ($'#1#$', $'#2#$', $'#3#$', $'#4#$', #5#, #6#, $'#7#$', $'#8#$', $'#9#$');';


// REPORT SCREEN FILTERING
slctCalibReportListByDate 	: STRING(5000) := 'SELECT TOP 100 CAST(ISNULL([ReportType], $'$') AS VARCHAR(50)) AS [ReportType], CAST(ISNULL([ReportID], $'$') AS VARCHAR(50)) AS [ReportID], CAST(ISNULL([CreatedOn], $'$') AS VARCHAR(30)) AS [CreatedOn], CAST(ISNULL([CreatedBy], $'$') AS VARCHAR(50)) AS [CreatedBy], CAST(ISNULL([Description], $'$') AS VARCHAR(200)) AS [Description], CAST(ISNULL([sPrimaryKey], $'$') AS VARCHAR(50)) AS [sPrimaryKey] FROM [dbo].[vw_ReportList_PumpCalibration] WHERE TRY_PARSE([CreatedOn] AS datetime USING $'en-GB$') >= #1# AND TRY_PARSE([CreatedOn] AS datetime USING $'en-GB$') <= #2# ORDER BY TRY_PARSE([CreatedOn] AS datetime USING $'en-GB$') DESC, CAST([ReportID] AS INT) DESC;';
slctSystemSettingsReportListByDate : STRING(5000) := 'SELECT TOP 100 CAST(ISNULL([ReportType], $'$') AS VARCHAR(50)) AS [ReportType], CAST(ISNULL([ReportID], $'$') AS VARCHAR(50)) AS [ReportID], CAST(ISNULL([CreatedOn], $'$') AS VARCHAR(30)) AS [CreatedOn], CAST(ISNULL([CreatedBy], $'$') AS VARCHAR(50)) AS [CreatedBy], CAST(ISNULL([Description], $'$') AS VARCHAR(200)) AS [Description], CAST(ISNULL([sPrimaryKey], $'$') AS VARCHAR(50)) AS [sPrimaryKey] FROM [dbo].[vw_ReportList_SystemSettings] WHERE TRY_PARSE([CreatedOn] AS datetime USING $'en-GB$') >= #1# AND TRY_PARSE([CreatedOn] AS datetime USING $'en-GB$') <= #2# ORDER BY TRY_PARSE([CreatedOn] AS datetime USING $'en-GB$') DESC, CAST([ReportID] AS INT) DESC;';
slctMethodReportSearchLatestByDate : STRING(5000) := 'SELECT TOP 100 CAST(ISNULL([ReportType], $'$') AS VARCHAR(50)) AS [ReportType], CAST(ISNULL([ReportID], $'$') AS VARCHAR(50)) AS [ReportID], CAST(ISNULL([CreatedOn], $'$') AS VARCHAR(30)) AS [CreatedOn], CAST(ISNULL([CreatedBy], $'$') AS VARCHAR(50)) AS [CreatedBy], CAST(ISNULL([Description], $'$') AS VARCHAR(200)) AS [Description], CAST(ISNULL([sPrimaryKey], $'$') AS VARCHAR(50)) AS [sPrimaryKey] FROM [dbo].[vw_ReportList_Recipe] WHERE TRY_PARSE(REPLACE([CreatedOn], $'D#$', $'$') AS datetime USING $'en-GB$') >= #1# AND TRY_PARSE(REPLACE([CreatedOn], $'D#$', $'$') AS datetime USING $'en-GB$') <= #2# ORDER BY TRY_PARSE(REPLACE([CreatedOn], $'D#$', $'$') AS datetime USING $'en-GB$') DESC, CAST([ReportID] AS INT) DESC;';
slctLinearReportListByDate 	: STRING(5000) := 'SELECT TOP 100 CAST(ISNULL([ReportType], $'$') AS VARCHAR(50)) AS [ReportType], CAST(ISNULL([ReportID], $'$') AS VARCHAR(50)) AS [ReportID], CAST(ISNULL([CreatedOn], $'$') AS VARCHAR(30)) AS [CreatedOn], CAST(ISNULL([CreatedBy], $'$') AS VARCHAR(50)) AS [CreatedBy], CAST(ISNULL([Description], $'$') AS VARCHAR(200)) AS [Description], CAST(ISNULL([sPrimaryKey], $'$') AS VARCHAR(50)) AS [sPrimaryKey] FROM [dbo].[vw_ReportList_Linear] WHERE TRY_PARSE([CreatedOn] AS datetime USING $'en-GB$') >= #1# AND TRY_PARSE([CreatedOn] AS datetime USING $'en-GB$') <= #2# ORDER BY TRY_PARSE([CreatedOn] AS datetime USING $'en-GB$') DESC, CAST([ReportID] AS INT) DESC;';
slctLinearHistoryReport 	: STRING(5000) := 'SELECT TOP 200 ISNULL([ID_Linear], 0) AS [ID_Linear], CAST(ISNULL([pump1], $'$') AS VARCHAR(100)) AS [pump1], CAST(ISNULL([pump2], $'$') AS VARCHAR(100)) AS [pump2], CAST(ISNULL([pump3], $'$') AS VARCHAR(100)) AS [pump3], CAST(ISNULL([pump4], $'$') AS VARCHAR(100)) AS [pump4], CAST(ISNULL([pump5], $'$') AS VARCHAR(100)) AS [pump5], CAST(ISNULL([pump6], $'$') AS VARCHAR(100)) AS [pump6], CAST(ISNULL([pump7], $'$') AS VARCHAR(100)) AS [pump7], CAST(ISNULL([pump8], $'$') AS VARCHAR(100)) AS [pump8], CAST(ISNULL([pump9], $'$') AS VARCHAR(100)) AS [pump9], CAST(ISNULL([pump10], $'$') AS VARCHAR(100)) AS [pump10], CAST(ISNULL([changedBy], $'$') AS VARCHAR(100)) AS [changedBy], CAST(ISNULL([changedOn], $'$') AS VARCHAR(100)) AS [changedOn] FROM [dbo].[LINEAR] ORDER BY [ID_Linear] DESC;';

//CURRENT REPORTS
slctLastLinear 	: STRING(5000) := 'SELECT TOP 1 ISNULL([ID_Linear], 0) AS [ID_Linear], CAST(ISNULL([pump1], $'$') AS VARCHAR(100)) AS [pump1], CAST(ISNULL([pump2], $'$') AS VARCHAR(100)) AS [pump2], CAST(ISNULL([pump3], $'$') AS VARCHAR(100)) AS [pump3], CAST(ISNULL([pump4], $'$') AS VARCHAR(100)) AS [pump4], CAST(ISNULL([pump5], $'$') AS VARCHAR(100)) AS [pump5], CAST(ISNULL([pump6], $'$') AS VARCHAR(100)) AS [pump6], CAST(ISNULL([pump7], $'$') AS VARCHAR(100)) AS [pump7], CAST(ISNULL([pump8], $'$') AS VARCHAR(100)) AS [pump8], CAST(ISNULL([pump9], $'$') AS VARCHAR(100)) AS [pump9], CAST(ISNULL([pump10], $'$') AS VARCHAR(100)) AS [pump10], CAST(ISNULL([changedBy], $'$') AS VARCHAR(100)) AS [changedBy], CAST(ISNULL([changedOn], $'$') AS VARCHAR(100)) AS [changedOn] FROM [dbo].[LINEAR] ORDER BY [ID_Linear] DESC;';
slctLastRun		: STRING(1000) := 'SELECT TOP 1 [runNo], [analyst], [comment], [softwareVersion], [sysMasterRevision], [sysSettingsRevision], [meterVelocity], [runVelocity], [emptyTubesFactor], [fillTubesFactor], [solvent1NameRevision], [solvent2NameRevision], [solvent3NameRevision], [solvent4NameRevision], [timeEventStarted], [timeEventCompleted], [methodID], [CalibrationNo] FROM [dbo].[RUNS] ORDER BY [runNo] DESC;';

(******************************************************************************************************)

(***** Pump Calibration Report Variables **************************************************************)

bBuildPCR			: BOOL;
stParameter_PCR		: ST_Parameters_PCR;
astData_PCR	  		: ARRAY[1..100] OF ST_Data_PCR;
lastCalibID			: ARRAY[0..1] OF INT;
lastCalibData		: array[1..100] of ST_Data_PCR;


(******************************************************************************************************)
	
(***** Post-Run Report Variables **********************************************************************)

bBuildPRRW		: BOOL;
stPostRunReport	: ARRAY[0..5] OF ST_PostRunReport;
lastRunID		: ARRAY[0..1] OF INT;
stPostRunInfo	: ST_PostRunReport;
runIsDone		: BOOL;

(******************************************************************************************************)

(***** User History Report Variables ******************************************************************)

bBuildUHR	   : BOOL;
astData_UHR	   : ARRAY[0..100] OF ST_Data_UHR;

(******************************************************************************************************)

(***** Current Users List Variables *****************************************************************)

bBuildCUL	   : BOOL;
astData_CUL	   : ARRAY[0..1000] OF ST_Data_CUL;

(******************************************************************************************************)

(***** Method Report Variables ************************************************************************)

bBuildMR			: BOOL;
stParameter_MR		: ST_Parameters_MR;
astVolData			: ARRAY[1..10] OF ST_VolumeData;
listOfMethod		: ARRAY[1..500] OF ST_ListMethod;
methodName			: STRING;
methodRevision		: STRING;
lastMethodID		: INT;
arrCompleteMethod	: ARRAY[1..100] OF ST_CompleteMethod;

(******************************************************************************************************)

(***** System Parameters Variables ********************************************************************)

stSysParameters	: ST_SysParameters;
listAllSystem	: ARRAY[0..500] OF ST_SysParameters;

(******************************************************************************************************)

(***** Solvents Variables *****************************************************************************)

stSolvents		: ST_Solvents;
listSolvents	: ARRAY[0..500] OF ST_Solvents;

(******************************************************************************************************)

(***** Linear Motors Variables *****************************************************************************)

stLinearMotors	: ST_LinearMotors;

(******************************************************************************************************)

(***** List Reports hmi *****************************************************************************)

aCalibReportList : ARRAY[1..100] OF ST_CalibrationReportListItem;

(******************************************************************************************************)

END_VAR

// ---- POUs/MARCO/OLD/GVL_Marco.TcGVL
{attribute 'qualified_only'}
VAR_GLOBAL
	
	enableAxi: ARRAY[1..10] OF BOOL;
	runFWD: ARRAY[1..10] OF BOOL;
	resetAxi: ARRAY[1..10] OF BOOL;
	revs: REAL;
	mL_target: REAL;
	runBWD: ARRAY[1..10] OF BOOL;
	enableValv: ARRAY[1..5] OF BOOL;
	valvPos: INT;
	calibResult: ARRAY[1..50] OF ST_Results;
	
END_VAR

// ---- POUs/MotionControl/IF_Actuator.TcIO
INTERFACE IF_Actuator
	//// Generic Interface for actuators

METHOD Disable : BOOL
VAR_INPUT
END_VAR
END_METHOD

METHOD Enable : BOOL
VAR_INPUT
END_VAR
END_METHOD

METHOD GetStatus : ST_ActuatorStatus
VAR_INPUT
END_VAR
END_METHOD

METHOD Reset : BOOL
VAR_INPUT
END_VAR
END_METHOD

END_INTERFACE

// ---- POUs/0. Main/MAIN_Control.TcPOU
PROGRAM MAIN_Control

VAR		
	bValveTest  : BOOL := FALSE;
	timerOnInit : TON;
    bLoadSysParametersExecute : BOOL;
    bLoadSysParametersReset   : BOOL;
END_VAR

timerOnInit(IN := TRUE, PT := T#10S);

//Main Controll
DB_Query();
PRG_MasterControl();
PRG_UpdateVariablesMoving();
PRG_SafetyHandle();
PRG_AxisAssignment();

//MainEvents
POU_EventTest();
POU_FaultHandler();
PRG_MasterSystemTime();

//MainHMI
PRG_HMIControl();
PRG_TowerAlarmLamps();
PRG_LevelHandler();
PRG_ValvePositionRecovery();

//MainServices
PRG_ReportsManager();
PRG_ShutdownPLC();
PRG_RecipeManager();
PRG_SystemInfo();
PRG_UserManagementHistory();

IF timerOnInit.Q
AND NOT DB_Load_SysParameters.bBusy
AND NOT DB_Load_SysParameters.bDone
AND NOT DB_Load_SysParameters.bError THEN
    bLoadSysParametersExecute := TRUE;
END_IF

DB_Load_SysParameters(
    bExecute := bLoadSysParametersExecute,
    bReset   := bLoadSysParametersReset
);

IF DB_Load_SysParameters.bDone OR DB_Load_SysParameters.bError THEN
    bLoadSysParametersExecute := FALSE;
END_IF

// Valve testing
IF bValveTest THEN
	PRG_ValveTest();
END_IF

END_PROGRAM

// ---- POUs/MARCO/DB/DB_Query.TcPOU
PROGRAM DB_Query
VAR_INPUT
	state: E_DB_QUERY_STATE;
	i: INT;
	j: INT;
END_VAR

VAR_OUTPUT
	bBusyDb : BOOL := FALSE;
END_VAR

VAR
	FB_SelectArray: FB_DBRecordArraySelect;
	FB_Insert: FB_DBRecordInsert_EX;
	cmd         : T_Maxstring := 'SELECT [ID], [userID], [accessLevel], [addDate], [enteredBy], [test] FROM [dbo].[TABLE01] ';
	insertString		: STRING(5000) := 'INSERT INTO [dbo].[TABLE01] ([NAME]) VALUES ( $'#1#$' )';
    (* Unter ARM*) 
    (*cmd       : T_Maxstring := 'SELECT ID,Timestamp,Value,Name FROM myTable'*)
    (*----------*)
    recordArray : ARRAY [1..5] OF ST_Data_CUL;
    busy        : BOOL;
    err         : BOOL;
    errid       : UDINT;
    sqlstate    : ST_DBSQLError;
    recAnz      : UDINT;
	bExecute	: BOOL;
	bExecute2	: BOOL;
	bExecuteIn	: BOOL;
	nome: STRING;
	cmdIn: STRING(10000);
	cmdSlc: STRING(10000);
	status: STRING;
	str: STRING;
	lastRunID: STRING;
	
	tempCmd: STRING(5000);
	timerVD: ton;
	start: BOOL;
	bDebug: BOOL;
	
	aPumpCalibHeader : ARRAY[1..1] OF ST_Parameters_PCR;
	bInitSelectCalibReportByID 			: BOOL := FALSE;
	bInitSelectCalibReportValuesByID	: BOOL := FALSE;
	bInitSelectSystemSettingsReportList : BOOL := FALSE;
	bInitSelectSystemSettingsByID       : BOOL := FALSE;
	bInitSelectCalibReportList			: BOOL := FALSE;
	bInitSelectMethodReportList			: BOOL := FALSE;
	bInitSelectMethodReportSearch		: BOOL := FALSE;
	bInitSelectRunReportList			: BOOL := FALSE;
	bInitSelectRecipeHeaderByID 		: BOOL := FALSE;
	bInitSelectRecipeVolumeByID 		: BOOL := FALSE;
	bInitSelectLinearByID 				: BOOL := FALSE;
	bInitSelectPostRunByID 				: BOOL := FALSE;
	bInitSelectPostRunMethodByID 		: BOOL := FALSE;
	bInitSelectPostRunVolumeByMethodID 	: BOOL := FALSE;
	bInitSelectLinearReportSearch 		: BOOL := FALSE;
	bInitSelectLastLinearReport 		: BOOL := FALSE;
	bInitSelectLastPostRunRun 			: BOOL := FALSE;
	bInitSelectLastPumpCalibration 		: BOOL := FALSE;
	bInitSelectSystemHistoryReport 		: BOOL := FALSE;
	bInitSelectLinearHistoryReport 		: BOOL := FALSE;
	bInitSelectCompleteMethodReport 	: BOOL := FALSE;
	bInitSelectCompleteMethodVolumes 	: BOOL := FALSE;
	iCompleteMethodIndex            	: INT := 1;
	sCompleteMethodID               	: STRING(20);
	
	sPostRunMethodID : STRING(20) := '';
	lastCalibID 	 : ARRAY[0..1] OF INT;
END_VAR

//FindAndReplace(pSrcString:= ADR(insertString), pDeleteString:= ADR('#1#'), pInsertString:= ADR(nome), pDstString:= ADR(cmdIn), nDstSize:= SIZEOF(cmdIn));	
timerVD();
Fill_Calibration_Data();
Fill_Method_Data();
DB_Load_CompleteMethod(start:= start);

bBusyDb := (state <> E_DB_QUERY_STATE.IDLE_STATE) AND (state <> E_DB_QUERY_STATE.ERROR_STATE);

IF timerVD.Q THEN
	state:= E_DB_QUERY_STATE.SELECT_VOLUME_DATA;
END_IF

CASE state OF
E_DB_QUERY_STATE.IDLE_STATE:
	
	state:= E_DB_QUERY_STATE.IDLE_STATE;
	FB_Insert(sNetID:= , hDBID:= 1, cbCmdSize:= SIZEOF(cmdIn), pCmdAddr:= ADR(cmdIn), bExecute:= FALSE, tTimeout:= T#15S, bBusy=> busy, bError=> err, nErrID=> errid, sSQLState=> sqlstate);
	FB_SelectArray(sNetID:= , hDBID:= 1, cbCmdSize:= SIZEOF(cmdSlc), pCmdAddr:= ADR(cmdSlc), nStartIndex:= 0, nRecordCount:= 1, cbRecordArraySize:= SIZEOF(GVL_DB.lastCalibID), pDestAddr:= ADR(GVL_DB.lastCalibID), bExecute:= FALSE, tTimeout:= T#15S, bBusy=> busy, bError=> err, nErrID=> errid, sSQLState=> sqlstate, nRecords=> recAnz);
		
E_DB_QUERY_STATE.SELECT_POST_LAST_RUN:
	
	FB_SelectArray(sNetID:= , hDBID:= 1, cbCmdSize:= SIZEOF(GVL_DB.slctLastRun), pCmdAddr:= ADR(GVL_DB.slctLastRun), nStartIndex:= 0, nRecordCount:= 5, cbRecordArraySize:= SIZEOF(GVL_DB.stPostRunReport), pDestAddr:= ADR(GVL_DB.stPostRunReport), bExecute:= TRUE, tTimeout:= T#15S, bBusy=> busy, bError=> err, nErrID=> errid, sSQLState=> sqlstate, nRecords=> recAnz);
	
	IF NOT FB_SelectArray.bBusy THEN
		state:= E_DB_QUERY_STATE.IDLE_STATE;
		bExecute:= FALSE;
	ELSIF FB_SelectArray.bError THEN	
		state:= E_DB_QUERY_STATE.ERROR_STATE;
	ELSE
		state:= E_DB_QUERY_STATE.SELECT_POST_LAST_RUN;
		bExecute:= FALSE;
	END_IF
	
E_DB_QUERY_STATE.INSERT_RUN:
	
	cmdIn:= GVL_DB.isrtRun;
	insertRunValues(start:=TRUE);
	FB_Insert(sNetID:= , hDBID:= 1, cbCmdSize:= SIZEOF(cmdIn), pCmdAddr:= ADR(cmdIn), bExecute:= TRUE, tTimeout:= T#15S, bBusy=> busy, bError=> err, nErrID=> errid, sSQLState=> sqlstate);
	
	IF NOT FB_Insert.bBusy THEN
		state:= E_DB_QUERY_STATE.IDLE_STATE;
		bExecuteIn:= FALSE;
	ELSIF FB_Insert.bError THEN	
		state:= E_DB_QUERY_STATE.ERROR_STATE;
	ELSE
		state:= E_DB_QUERY_STATE.INSERT_RUN;
		bExecuteIn:= FALSE;
	END_IF

E_DB_QUERY_STATE.SELECT_LAST_CALIBRATION_ID:
	
	FB_SelectArray(sNetID:= , hDBID:= 1, cbCmdSize:= SIZEOF(GVL_DB.slctLastCalibID), pCmdAddr:= ADR(GVL_DB.slctLastCalibID), nStartIndex:= 0, nRecordCount:= 1, cbRecordArraySize:= SIZEOF(GVL_DB.lastCalibID), pDestAddr:= ADR(GVL_DB.lastCalibID), bExecute:= TRUE, tTimeout:= T#15S, bBusy=> busy, bError=> err, nErrID=> errid, sSQLState=> sqlstate, nRecords=> recAnz);
	
	IF NOT FB_SelectArray.bBusy THEN
		state:= E_DB_QUERY_STATE.IDLE_STATE;
		bExecute:= FALSE;
	ELSIF FB_SelectArray.bError THEN	
		state:= E_DB_QUERY_STATE.ERROR_STATE;
	ELSE
		state:= E_DB_QUERY_STATE.SELECT_LAST_CALIBRATION_ID;
		bExecute:= FALSE;
	END_IF

E_DB_QUERY_STATE.SELECT_LAST_CALIBRATION:
	
	FB_SelectArray(sNetID:= , hDBID:= 1, cbCmdSize:= SIZEOF(GVL_DB.slctLastCalib), pCmdAddr:= ADR(GVL_DB.slctLastCalib), nStartIndex:= 0, nRecordCount:= 100, cbRecordArraySize:= SIZEOF(GVL_DB.lastCalibData), pDestAddr:= ADR(GVL_DB.lastCalibData), bExecute:= TRUE, tTimeout:= T#15S, bBusy=> busy, bError=> err, nErrID=> errid, sSQLState=> sqlstate, nRecords=> recAnz);
	
	IF NOT FB_SelectArray.bBusy THEN
		state:= E_DB_QUERY_STATE.IDLE_STATE;
		bExecute:= FALSE;
	ELSIF FB_SelectArray.bError THEN	
		state:= E_DB_QUERY_STATE.ERROR_STATE;
	ELSE
		state:= E_DB_QUERY_STATE.SELECT_LAST_CALIBRATION;
		bExecute:= FALSE;
	END_IF
	
E_DB_QUERY_STATE.INSERT_CALIBRATION_VALUES:

	cmdIn:= GVL_DB.isrtCalibValues;
	insertCalibValues(start:=TRUE, line:= GVL_Calibration.iResultIndex);
	FB_Insert(sNetID:= , hDBID:= 1, cbCmdSize:= SIZEOF(cmdIn), pCmdAddr:= ADR(cmdIn), bExecute:= TRUE, tTimeout:= T#15S, bBusy=> busy, bError=> err, nErrID=> errid, sSQLState=> sqlstate);
	
	IF NOT FB_Insert.bBusy THEN
		state:= E_DB_QUERY_STATE.IDLE_STATE;
		bExecuteIn:= FALSE;
	ELSIF FB_Insert.bError THEN	
		state:= E_DB_QUERY_STATE.ERROR_STATE;
	ELSE
		state:= E_DB_QUERY_STATE.INSERT_CALIBRATION_VALUES;
		bExecuteIn:= FALSE;
	END_IF

E_DB_QUERY_STATE.INSERT_CALIBRATION:

	cmdIn:= GVL_DB.isrtCalib;
	insertCalib(start:=TRUE);
	FB_Insert(sNetID:= , hDBID:= 1, cbCmdSize:= SIZEOF(cmdIn), pCmdAddr:= ADR(cmdIn), bExecute:= TRUE, tTimeout:= T#15S, bBusy=> busy, bError=> err, nErrID=> errid, sSQLState=> sqlstate);
	
	IF NOT FB_Insert.bBusy THEN
		state:= E_DB_QUERY_STATE.IDLE_STATE;
		bExecuteIn:= FALSE;
	ELSIF FB_Insert.bError THEN	
		state:= E_DB_QUERY_STATE.ERROR_STATE;
	ELSE
		state:= E_DB_QUERY_STATE.INSERT_CALIBRATION;
		//bExecuteIn:= FALSE;
	END_IF
	
// FIX: Delete an orphaned CALIBRATION_HEAD row when calibration is aborted
// before any measurement was recorded. Triggered from E_CalibStep.ERROR
// when iResultIndex <= 1. The CalibrationNo to delete is in stParameter_PCR.
// NOTE: Add DELETE_CALIBRATION_HEAD to E_DB_QUERY_STATE enum in your DUT.
E_DB_QUERY_STATE.DELETE_CALIBRATION_HEAD:

	cmdIn:= GVL_DB.dltCalibHead;
	deleteCalibHead(start:= TRUE);
	FB_Insert(sNetID:= , hDBID:= 1, cbCmdSize:= SIZEOF(cmdIn), pCmdAddr:= ADR(cmdIn), bExecute:= TRUE, tTimeout:= T#15S, bBusy => busy, bError => err, nErrID => errid, sSQLState => sqlstate);

	IF NOT FB_Insert.bBusy THEN
		state:= E_DB_QUERY_STATE.IDLE_STATE;
	ELSIF FB_Insert.bError THEN
		state:= E_DB_QUERY_STATE.ERROR_STATE;
	ELSE
		state:= E_DB_QUERY_STATE.DELETE_CALIBRATION_HEAD;
	END_IF
	
E_DB_QUERY_STATE.SELECT_LAST_SYSTEM_ID:
	
	FB_SelectArray(sNetID:= , hDBID:= 1, cbCmdSize:= SIZEOF(GVL_DB.slctLastSys), pCmdAddr:= ADR(GVL_DB.slctLastSys), nStartIndex:= 0, nRecordCount:= 1, cbRecordArraySize:= SIZEOF(GVL_DB.stSysParameters), pDestAddr:= ADR(GVL_DB.stSysParameters), bExecute:= TRUE, tTimeout:= T#15S, bBusy=> busy, bError=> err, nErrID=> errid, sSQLState=> sqlstate, nRecords=> recAnz);
	
	IF NOT FB_SelectArray.bBusy THEN
		state:= E_DB_QUERY_STATE.IDLE_STATE;
		bExecute:= FALSE;
	ELSIF FB_SelectArray.bError THEN	
		state:= E_DB_QUERY_STATE.ERROR_STATE;
	ELSE
		state:= E_DB_QUERY_STATE.SELECT_LAST_SYSTEM_ID;
		bExecute:= FALSE;
	END_IF	
	
E_DB_QUERY_STATE.SELECT_ALL_SYSTEM:
	
	FB_SelectArray(sNetID:= , hDBID:= 1, cbCmdSize:= SIZEOF(GVL_DB.slctAllSys), pCmdAddr:= ADR(GVL_DB.slctAllSys), nStartIndex:= 0, nRecordCount:= 1000, cbRecordArraySize:= SIZEOF(GVL_DB.listAllSystem), pDestAddr:= ADR(GVL_DB.listAllSystem), bExecute:= TRUE, tTimeout:= T#15S, bBusy=> busy, bError=> err, nErrID=> errid, sSQLState=> sqlstate, nRecords=> recAnz);
	
	IF NOT FB_SelectArray.bBusy THEN
		state:= E_DB_QUERY_STATE.IDLE_STATE;
		bExecute:= FALSE;
	ELSIF FB_SelectArray.bError THEN	
		state:= E_DB_QUERY_STATE.ERROR_STATE;
	ELSE
		state:= E_DB_QUERY_STATE.SELECT_ALL_SYSTEM;
		bExecute:= FALSE;
	END_IF
	
E_DB_QUERY_STATE.INSERT_SYS_PARAMETERS:

	cmdIn:= GVL_DB.isrtSys;
	insertSys(start:=TRUE);
	FB_Insert(sNetID:= , hDBID:= 1, cbCmdSize:= SIZEOF(cmdIn), pCmdAddr:= ADR(cmdIn), bExecute:= TRUE, tTimeout:= T#15S, bBusy=> busy, bError=> err, nErrID=> errid, sSQLState=> sqlstate);
	
	IF NOT FB_Insert.bBusy THEN
		state:= E_DB_QUERY_STATE.IDLE_STATE;
		bExecuteIn:= FALSE;
	ELSIF FB_Insert.bError THEN	
		state:= E_DB_QUERY_STATE.ERROR_STATE;
	ELSE
		state:= E_DB_QUERY_STATE.INSERT_SYS_PARAMETERS;
		//bExecuteIn:= FALSE;
	END_IF	

E_DB_QUERY_STATE.SELECT_ALL_METHODS:
	
